KUKA KRL program: MyProgram_264().src

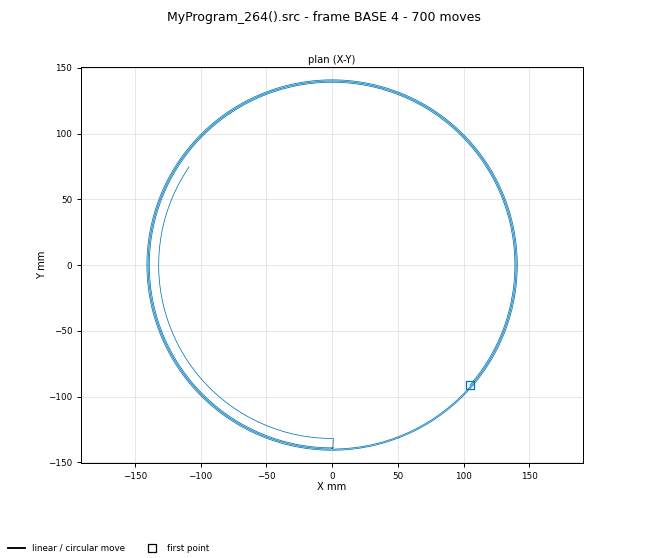
[picture p0: tool path of MyProgram_264().src in frame BASE 4, 700 of 700 moves have a stored position in this frame; points joined in program order, loops and branches not executed]
&ACCESS RVP
&REL 1
&PARAM TEMPLATE = C:\KRC\Roboter\Template\vorgabe
&PARAM EDITMASK = *
DEF MyProgram_264()
; ---- Setting reference (Base) ----
$BASE = BASE_DATA[4]

; --------------------------
; ---- Setting tool (TCP) ----
$TOOL = TOOL_DATA[3]
; --------------------------

$VEL.CP = VEL_APROX_PRINT
Startdeposition()
$VEL.CP = VEL_PRINT
LIN {X 104.7869,Y -91.2895,Z 168,A -38.7175,B 9.9687,C 0.2931,E1 10.0953,E2 489.8087} C_DIS
LIN {X 108.3715,Y -87.0044,Z 168,A -36.6212,B 9.9688,C 0.2929,E1 10.0989,E2 487.737} C_DIS
LIN {X 111.1205,Y -83.4649,Z 168,A -34.5628,B 9.9691,C 0.2832,E1 10.1024,E2 485.6491} C_DIS
LIN {X 113.1517,Y -80.6895,Z 168,A -32.7499,B 9.9694,C 0.2697,E1 10.1055,E2 483.7829} C_DIS
LIN {X 116.399,Y -75.9304,Z 168,A -31.0627,B 9.9691,C 0.2812,E1 10.1079,E2 482.1831} C_DIS
LIN {X 118.3407,Y -72.8666,Z 168,A -29.4296,B 9.9693,C 0.2739,E1 10.1104,E2 480.5305} C_DIS
LIN {X 120.9717,Y -68.4109,Z 168,A -27.417,B 9.9694,C 0.2715,E1 10.1131,E2 478.5313} C_DIS
LIN {X 123.1966,Y -64.3133,Z 168,A -24.8855,B 9.9699,C 0.2509,E1 10.1165,E2 475.918} C_DIS
LIN {X 125.8704,Y -58.9115,Z 168,A -23.1595,B 9.9696,C 0.2636,E1 10.1185,E2 474.2886} C_DIS
LIN {X 127.3983,Y -55.528,Z 168,A -21.7568,B 9.9696,C 0.2626,E1 10.1201,E2 472.9008} C_DIS
LIN {X 128.707,Y -52.4242,Z 168,A -20.3371,B 9.9698,C 0.2581,E1 10.1216,E2 471.4756} C_DIS
LIN {X 130.4635,Y -47.89,Z 168,A -18.2188,B 9.97,C 0.2496,E1 10.1237,E2 469.3404} C_DIS
LIN {X 131.6831,Y -44.4232,Z 168,A -16.8072,B 9.97,C 0.248,E1 10.125,E2 467.9405} C_DIS
LIN {X 132.7574,Y -41.1001,Z 168,A -15.3867,B 9.97,C 0.2445,E1 10.1262,E2 466.521} C_DIS
LIN {X 134.004,Y -36.8358,Z 168,A -13.5572,B 9.9702,C 0.2393,E1 10.1276,E2 464.6898} C_DIS
LIN {X 135.3311,Y -31.6154,Z 168,A -11.3086,B 9.9704,C 0.2323,E1 10.1291,E2 462.4352} C_DIS
LIN {X 136.0558,Y -28.3338,Z 168,A -9.341,B 9.9708,C 0.2134,E1 10.1302,E2 460.3905} C_DIS
LIN {X 137.1037,Y -22.7202,Z 168,A -8.0736,B 9.9703,C 0.2343,E1 10.1308,E2 459.2616} C_DIS
LIN {X 137.4864,Y -20.2859,Z 168,A -6.7394,B 9.9706,C 0.2233,E1 10.1313,E2 457.8854} C_DIS
LIN {X 137.9944,Y -16.4673,Z 168,A -5.1719,B 9.9706,C 0.2192,E1 10.1319,E2 456.3189} C_DIS
LIN {X 138.5607,Y -10.7209,Z 168,A -2.595,B 9.9709,C 0.2073,E1 10.1325,E2 453.7142} C_DIS
LIN {X 138.8592,Y -5.6425,Z 168,A -0.7367,B 9.9709,C 0.2073,E1 10.1328,E2 451.8846} C_DIS
LIN {X 138.9611,Y -1.9096,Z 168,A 0.6796,B 9.9709,C 0.2059,E1 10.1328,E2 450.4827} C_DIS
LIN {X 138.9263,Y 3.6331,Z 168,A 3.0218,B 9.9711,C 0.1978,E1 10.1328,E2 448.1311} C_DIS
LIN {X 138.6111,Y 10.0308,Z 168,A 5.6741,B 9.9713,C 0.1898,E1 10.1324,E2 445.4748} C_DIS
LIN {X 138.3396,Y 13.2584,Z 168,A 7.4808,B 9.9716,C 0.1739,E1 10.1319,E2 443.606} C_DIS
LIN {X 137.7917,Y 18.0849,Z 168,A 8.8238,B 9.9714,C 0.1849,E1 10.1314,E2 442.3462} C_DIS
LIN {X 137.0969,Y 22.761,Z 168,A 10.9205,B 9.9715,C 0.1756,E1 10.1305,E2 440.2289} C_DIS
LIN {X 136.0747,Y 28.2409,Z 168,A 13.3844,B 9.9717,C 0.1648,E1 10.1292,E2 437.7417} C_DIS
LIN {X 135.321,Y 31.66,Z 168,A 14.6274,B 9.9717,C 0.1658,E1 10.1284,E2 436.5233} C_DIS
LIN {X 134.3492,Y 35.5518,Z 168,A 16.1439,B 9.9717,C 0.1646,E1 10.1273,E2 435.023} C_DIS
LIN {X 133.4563,Y 38.7692,Z 168,A 17.4893,B 9.9717,C 0.1616,E1 10.1263,E2 433.6804} C_DIS
LIN {X 132.3926,Y 42.2583,Z 168,A 18.9598,B 9.9718,C 0.1582,E1 10.1251,E2 432.213} C_DIS
LIN {X 131.3467,Y 45.405,Z 168,A 20.2249,B 9.9718,C 0.157,E1 10.124,E2 430.9599} C_DIS
LIN {X 130.5672,Y 47.6024,Z 168,A 21.8935,B 9.9721,C 0.1366,E1 10.1223,E2 429.1998} C_DIS
LIN {X 128.6889,Y 52.4691,Z 168,A 23.0407,B 9.9719,C 0.156,E1 10.1212,E2 428.1795} C_DIS
LIN {X 127.1442,Y 56.1102,Z 168,A 25.0796,B 9.9721,C 0.1415,E1 10.1189,E2 426.0876} C_DIS
LIN {X 125.5425,Y 59.6045,Z 168,A 26.6572,B 9.9721,C 0.1375,E1 10.1171,E2 424.5098} C_DIS
LIN {X 123.808,Y 63.1275,Z 168,A 28.1243,B 9.9721,C 0.1371,E1 10.1152,E2 423.061} C_DIS
LIN {X 122.1696,Y 66.2478,Z 168,A 29.4062,B 9.9721,C 0.1377,E1 10.1136,E2 421.8} C_DIS
LIN {X 119.9358,Y 70.2099,Z 168,A 31.3397,B 9.9721,C 0.1316,E1 10.1109,E2 419.858} C_DIS
LIN {X 117.6886,Y 73.9159,Z 168,A 33.3363,B 9.9723,C 0.122,E1 10.1079,E2 417.8337} C_DIS
LIN {X 115.2813,Y 77.6165,Z 168,A 35.1156,B 9.9723,C 0.1186,E1 10.1052,E2 416.0585} C_DIS
LIN {X 112.6825,Y 81.3436,Z 168,A 36.9745,B 9.9724,C 0.1146,E1 10.1022,E2 414.2005} C_DIS
LIN {X 110.8525,Y 83.8201,Z 168,A 38.4939,B 9.9725,C 0.1055,E1 10.0996,E2 412.6485} C_DIS
LIN {X 108.4731,Y 86.8782,Z 168,A 39.6916,B 9.9725,C 0.1117,E1 10.0976,E2 411.5011} C_DIS
LIN {X 105.8164,Y 90.0942,Z 168,A 41.4849,B 9.9725,C 0.1061,E1 10.0944,E2 409.6976} C_DIS
LIN {X 99.6435,Y 96.8779,Z 168,A 45.2327,B 9.9725,C 0.099,E1 10.0873,E2 405.9528} C_DIS
LIN {X 97.1213,Y 99.4061,Z 168,A 46.8412,B 9.9726,C 0.0928,E1 10.084,E2 404.3264} C_DIS
LIN {X 93.1563,Y 103.1313,Z 168,A 48.9073,B 9.9726,C 0.0927,E1 10.0798,E2 402.2821} C_DIS
LIN {X 90.6095,Y 105.3754,Z 168,A 50.6855,B 9.9727,C 0.0809,E1 10.076,E2 400.4553} C_DIS
LIN {X 87.221,Y 108.1968,Z 168,A 52.1284,B 9.9727,C 0.0867,E1 10.0729,E2 399.0597} C_DIS
LIN {X 83.4306,Y 111.1464,Z 168,A 53.8675,B 9.9727,C 0.089,E1 10.0691,E2 397.3507} C_DIS
LIN {X 81.247,Y 112.7524,Z 168,A 55.195,B 9.9727,C 0.0821,E1 10.0661,E2 395.9964} C_DIS
LIN {X 77.5243,Y 115.344,Z 168,A 57.0601,B 9.9727,C 0.0792,E1 10.0618,E2 394.1316} C_DIS
LIN {X 73.7727,Y 117.7787,Z 168,A 58.8556,B 9.9727,C 0.0775,E1 10.0575,E2 392.3419} C_DIS
LIN {X 70.011,Y 120.053,Z 168,A 60.6788,B 9.9727,C 0.0746,E1 10.0532,E2 390.5172} C_DIS
LIN {X 66.8198,Y 121.8576,Z 168,A 62.1695,B 9.9727,C 0.073,E1 10.0495,E2 389.029} C_DIS
LIN {X 61.3179,Y 124.7143,Z 168,A 64.57,B 9.9727,C 0.0734,E1 10.0436,E2 386.6479} C_DIS
LIN {X 58.4874,Y 126.0665,Z 168,A 65.8378,B 9.9727,C 0.0724,E1 10.0404,E2 385.3833} C_DIS
LIN {X 55.3605,Y 127.4707,Z 168,A 67.2727,B 9.9728,C 0.0703,E1 10.0367,E2 383.9457} C_DIS
LIN {X 52.2262,Y 128.7868,Z 168,A 68.6604,B 9.9728,C 0.0691,E1 10.0332,E2 382.5599} C_DIS
LIN {X 48.8963,Y 130.0873,Z 168,A 70.0927,B 9.9728,C 0.0685,E1 10.0294,E2 381.1329} C_DIS
LIN {X 45.7955,Y 131.2113,Z 168,A 71.5098,B 9.9728,C 0.0659,E1 10.0257,E2 379.7088} C_DIS
LIN {X 42.4601,Y 132.3281,Z 168,A 72.9338,B 9.9728,C 0.0653,E1 10.0219,E2 378.2882} C_DIS
LIN {X 39.2358,Y 133.3197,Z 168,A 74.1058,B 9.9728,C 0.0691,E1 10.0189,E2 377.1439} C_DIS
LIN {X 35.492,Y 134.3651,Z 168,A 76.3709,B 9.9729,C 0.0529,E1 10.0125,E2 374.7958} C_DIS
LIN {X 31.4057,Y 135.3791,Z 168,A 77.701,B 9.9729,C 0.061,E1 10.0091,E2 373.5173} C_DIS
LIN {X 27.0023,Y 136.3268,Z 168,A 80.0388,B 9.9729,C 0.0492,E1 10.0025,E2 371.1194} C_DIS
LIN {X 22.5072,Y 137.1392,Z 168,A 81.6679,B 9.9729,C 0.0541,E1 9.9981,E2 369.5229} C_DIS
LIN {X 19.253,Y 137.634,Z 168,A 82.8687,B 9.9729,C 0.057,E1 9.9948,E2 368.3422} C_DIS
LIN {X 15.4145,Y 138.1171,Z 168,A 84.8657,B 9.9729,C 0.0477,E1 9.9892,E2 366.2951} C_DIS
LIN {X 10.7583,Y 138.558,Z 168,A 86.4757,B 9.9729,C 0.0543,E1 9.9848,E2 364.726} C_DIS
LIN {X 5.6517,Y 138.8588,Z 168,A 88.4161,B 9.9729,C 0.0578,E1 9.9794,E2 362.8077} C_DIS
LIN {X 1.3259,Y 138.9685,Z 168,A 90.5444,B 9.9729,C 0.0503,E1 9.9734,E2 360.6369} C_DIS
LIN {X -2.4839,Y 138.9515,Z 168,A 91.9187,B 9.9729,C 0.0547,E1 9.9696,E2 359.288} C_DIS
LIN {X -7.6751,Y 138.7632,Z 168,A 94.0131,B 9.9729,C 0.0561,E1 9.9638,E2 357.2007} C_DIS
LIN {X -11.7705,Y 138.4742,Z 168,A 96.3131,B 9.9729,C 0.0434,E1 9.9572,E2 354.8249} C_DIS
LIN {X -17.6085,Y 137.8542,Z 168,A 98.4749,B 9.9729,C 0.0499,E1 9.9513,E2 352.6973} C_DIS
LIN {X -22.0537,Y 137.2147,Z 168,A 99.978,B 9.9729,C 0.0583,E1 9.9473,E2 351.2392} C_DIS
LIN {X -26.5941,Y 136.406,Z 168,A 101.7752,B 9.9729,C 0.0616,E1 9.9424,E2 349.4562} C_DIS
LIN {X -30.5737,Y 135.5691,Z 168,A 103.454,B 9.9729,C 0.0626,E1 9.9378,E2 347.7783} C_DIS
LIN {X -34.2317,Y 134.6914,Z 168,A 104.9802,B 9.9729,C 0.0643,E1 9.9336,E2 346.2561} C_DIS
LIN {X -37.445,Y 133.8336,Z 168,A 106.4119,B 9.9729,C 0.0641,E1 9.9298,E2 344.8179} C_DIS
LIN {X -40.4898,Y 132.9442,Z 168,A 108.0789,B 9.9729,C 0.0578,E1 9.9252,E2 343.1067} C_DIS
LIN {X -44.2338,Y 131.7461,Z 168,A 109.3437,B 9.9729,C 0.0667,E1 9.922,E2 341.8879} C_DIS
LIN {X -48.1285,Y 130.3749,Z 168,A 110.9864,B 9.9729,C 0.0697,E1 9.9177,E2 340.2539} C_DIS
LIN {X -51.4358,Y 129.1054,Z 168,A 112.3928,B 9.9728,C 0.0724,E1 9.914,E2 338.8554} C_DIS
LIN {X -55.5497,Y 127.3889,Z 168,A 114.4516,B 9.9728,C 0.0701,E1 9.9087,E2 336.7705} C_DIS
LIN {X -59.5895,Y 125.5497,Z 168,A 116.094,B 9.9728,C 0.0762,E1 9.9046,E2 335.153} C_DIS
LIN {X -62.3414,Y 124.2079,Z 168,A 117.6958,B 9.9728,C 0.071,E1 9.9005,E2 333.5099} C_DIS
LIN {X -66.1173,Y 122.2404,Z 168,A 119.509,B 9.9728,C 0.0723,E1 9.896,E2 331.691} C_DIS
LIN {X -68.9786,Y 120.6484,Z 168,A 120.6619,B 9.9728,C 0.0783,E1 9.8933,E2 330.564} C_DIS
LIN {X -71.4953,Y 119.1748,Z 168,A 122.3694,B 9.9728,C 0.07,E1 9.8891,E2 328.7941} C_DIS
LIN {X -75.6051,Y 116.6102,Z 168,A 123.715,B 9.9727,C 0.0863,E1 9.8861,E2 327.5322} C_DIS
LIN {X -78.7988,Y 114.4764,Z 168,A 125.4857,B 9.9727,C 0.0852,E1 9.8819,E2 325.7395} C_DIS
LIN {X -82.4494,Y 111.8758,Z 168,A 127.1228,B 9.9727,C 0.0926,E1 9.8783,E2 324.1305} C_DIS
LIN {X -86.4838,Y 108.7871,Z 168,A 129.6992,B 9.9727,C 0.0869,E1 9.8725,E2 321.4958} C_DIS
LIN {X -89.1735,Y 106.5935,Z 168,A 130.916,B 9.9727,C 0.0938,E1 9.8699,E2 320.3074} C_DIS
LIN {X -92.5782,Y 103.6502,Z 168,A 132.755,B 9.9726,C 0.0978,E1 9.8661,E2 318.4723} C_DIS
LIN {X -96.5219,Y 99.9881,Z 168,A 135.3869,B 9.9726,C 0.0942,E1 9.8606,E2 315.7907} C_DIS
LIN {X -99.4725,Y 97.0537,Z 168,A 136.7519,B 9.9726,C 0.1047,E1 9.8581,E2 314.4716} C_DIS
LIN {X -102.5413,Y 93.8054,Z 168,A 138.3633,B 9.9724,C 0.1132,E1 9.8551,E2 312.891} C_DIS
LIN {X -105.8315,Y 90.0764,Z 168,A 141.0491,B 9.9725,C 0.1054,E1 9.85,E2 310.1276} C_DIS
LIN {X -108.4461,Y 86.9114,Z 168,A 142.4577,B 9.9725,C 0.1149,E1 9.8476,E2 308.7565} C_DIS
LIN {X -110.6702,Y 84.0616,Z 168,A 143.8995,B 9.9724,C 0.1193,E1 9.8452,E2 307.3224} C_DIS
LIN {X -113.7992,Y 79.7744,Z 168,A 146.1492,B 9.9724,C 0.1234,E1 9.8415,E2 305.0674} C_DIS
LIN {X -116.3521,Y 76.0026,Z 168,A 148.054,B 9.9723,C 0.1275,E1 9.8385,E2 303.1611} C_DIS
LIN {X -118.6956,Y 72.2884,Z 168,A 149.9103,B 9.9723,C 0.1311,E1 9.8358,E2 301.3011} C_DIS
LIN {X -120.9843,Y 68.3884,Z 168,A 151.8068,B 9.9722,C 0.1353,E1 9.8332,E2 299.4025} C_DIS
LIN {X -123.1081,Y 64.4819,Z 168,A 153.8724,B 9.9722,C 0.1356,E1 9.8304,E2 297.3095} C_DIS
LIN {X -124.7232,Y 61.2998,Z 168,A 155.1789,B 9.972,C 0.1426,E1 9.8288,E2 296.0254} C_DIS
LIN {X -127.0073,Y 56.4162,Z 168,A 157.3275,B 9.972,C 0.15,E1 9.8264,E2 293.8885} C_DIS
LIN {X -128.5481,Y 52.8162,Z 168,A 159.4017,B 9.972,C 0.1457,E1 9.8241,E2 291.7581} C_DIS
LIN {X -130.0853,Y 48.9017,Z 168,A 160.672,B 9.9718,C 0.1592,E1 9.8229,E2 290.5482} C_DIS
LIN {X -132.1241,Y 43.0961,Z 168,A 163.3195,B 9.9718,C 0.1642,E1 9.8205,E2 287.8896} C_DIS
LIN {X -133.3063,Y 39.2816,Z 168,A 164.9105,B 9.9716,C 0.1699,E1 9.8192,E2 286.3072} C_DIS
LIN {X -134.2142,Y 36.058,Z 168,A 166.3635,B 9.9716,C 0.1724,E1 9.8181,E2 284.8466} C_DIS
LIN {X -135.0793,Y 32.6675,Z 168,A 167.7655,B 9.9715,C 0.1773,E1 9.8172,E2 283.4512} C_DIS
LIN {X -135.8366,Y 29.3601,Z 168,A 169.1877,B 9.9715,C 0.1809,E1 9.8163,E2 282.0276} C_DIS
LIN {X -136.4454,Y 26.388,Z 168,A 170.5451,B 9.9715,C 0.1825,E1 9.8156,E2 280.6581} C_DIS
LIN {X -137.1353,Y 22.5308,Z 168,A 172.1893,B 9.9713,C 0.1866,E1 9.8148,E2 279.0119} C_DIS
LIN {X -137.7668,Y 18.2749,Z 168,A 173.9456,B 9.9713,C 0.1921,E1 9.8141,E2 277.2597} C_DIS
LIN {X -138.1801,Y 14.8292,Z 168,A 175.3528,B 9.9711,C 0.1967,E1 9.8137,E2 275.8569} C_DIS
LIN {X -138.6204,Y 9.9036,Z 168,A 177.2102,B 9.971,C 0.206,E1 9.8133,E2 274.0245} C_DIS
LIN {X -138.8726,Y 5.2979,Z 168,A 179.3932,B 9.971,C 0.2063,E1 9.813,E2 271.8079} C_DIS
LIN {X -138.9511,Y 2.5119,Z 168,A -178.8031,B 9.9711,C 0.1973,E1 9.8129,E2 269.9221} C_DIS
LIN {X -138.9457,Y -2.8364,Z 168,A -177.2929,B 9.9707,C 0.2169,E1 9.8129,E2 268.5026} C_DIS
LIN {X -138.7047,Y -8.6416,Z 168,A -174.7671,B 9.9707,C 0.2214,E1 9.8133,E2 265.9626} C_DIS
LIN {X -138.3646,Y -12.9984,Z 168,A -172.9482,B 9.9705,C 0.2263,E1 9.8137,E2 264.1432} C_DIS
LIN {X -137.9891,Y -16.5116,Z 168,A -171.4819,B 9.9705,C 0.2303,E1 9.8141,E2 262.677} C_DIS
LIN {X -137.4533,Y -20.5131,Z 168,A -169.6739,B 9.9704,C 0.2324,E1 9.8149,E2 260.8524} C_DIS
LIN {X -136.8786,Y -24.0426,Z 168,A -168.2662,B 9.9703,C 0.2379,E1 9.8155,E2 259.4545} C_DIS
LIN {X -136.2873,Y -27.1964,Z 168,A -166.9044,B 9.9702,C 0.2409,E1 9.8163,E2 258.0889} C_DIS
LIN {X -135.5229,Y -30.7758,Z 168,A -165.4066,B 9.9701,C 0.2454,E1 9.8172,E2 256.5938} C_DIS
LIN {X -134.672,Y -34.308,Z 168,A -163.9032,B 9.97,C 0.2495,E1 9.8182,E2 255.0909} C_DIS
LIN {X -133.92,Y -37.1362,Z 168,A -162.3001,B 9.97,C 0.2453,E1 9.8194,E2 253.4382} C_DIS
LIN {X -132.8591,Y -40.768,Z 168,A -161.1109,B 9.9698,C 0.2567,E1 9.8203,E2 252.2976} C_DIS
LIN {X -131.6541,Y -44.5101,Z 168,A -159.3701,B 9.9698,C 0.2588,E1 9.8219,E2 250.5428} C_DIS
LIN {X -130.2278,Y -48.5213,Z 168,A -157.5157,B 9.9697,C 0.2617,E1 9.8236,E2 248.6771} C_DIS
LIN {X -128.3545,Y -53.2798,Z 168,A -155.5113,B 9.9695,C 0.2693,E1 9.8257,E2 246.6875} C_DIS
LIN {X -126.9695,Y -56.5007,Z 168,A -154.0901,B 9.9693,C 0.2736,E1 9.8273,E2 245.2705} C_DIS
LIN {X -125.5352,Y -59.6198,Z 168,A -152.6233,B 9.9693,C 0.2763,E1 9.8291,E2 243.798} C_DIS
LIN {X -124.0044,Y -62.7419,Z 168,A -151.1771,B 9.9692,C 0.2797,E1 9.8309,E2 242.3512} C_DIS
LIN {X -122.2078,Y -66.1778,Z 168,A -149.4378,B 9.9692,C 0.281,E1 9.8332,E2 240.595} C_DIS
LIN {X -119.9592,Y -70.1707,Z 168,A -147.5406,B 9.969,C 0.2855,E1 9.8358,E2 238.698} C_DIS
LIN {X -117.5827,Y -74.0837,Z 168,A -145.6598,B 9.9689,C 0.2902,E1 9.8386,E2 236.8191} C_DIS
LIN {X -115.2184,Y -77.71,Z 168,A -143.8229,B 9.9688,C 0.2935,E1 9.8414,E2 234.9765} C_DIS
LIN {X -112.5662,Y -81.5042,Z 168,A -142.027,B 9.9686,C 0.3001,E1 9.8443,E2 233.1961} C_DIS
LIN {X -110.0316,Y -84.8953,Z 168,A -140.3109,B 9.9685,C 0.3046,E1 9.8472,E2 231.4847} C_DIS
LIN {X -107.8706,Y -87.6252,Z 168,A -138.6725,B 9.9685,C 0.3038,E1 9.8501,E2 229.8208} C_DIS
LIN {X -103.7204,Y -92.4993,Z 168,A -135.7389,B 9.9685,C 0.3035,E1 9.8555,E2 226.8505} C_DIS
LIN {X -101.1547,Y -95.2985,Z 168,A -134.4399,B 9.9682,C 0.3121,E1 9.858,E2 225.5864} C_DIS
LIN {X -97.8845,Y -98.6544,Z 168,A -132.4981,B 9.9682,C 0.3157,E1 9.8618,E2 223.644} C_DIS
LIN {X -94.6627,Y -101.7499,Z 168,A -130.6386,B 9.968,C 0.3189,E1 9.8655,E2 221.783} C_DIS
LIN {X -91.8147,Y -104.3272,Z 168,A -128.9762,B 9.968,C 0.3202,E1 9.869,E2 220.1109} C_DIS
LIN {X -88.6264,Y -107.0487,Z 168,A -127.3089,B 9.9678,C 0.3246,E1 9.8726,E2 218.4519} C_DIS
LIN {X -85.2071,Y -109.7899,Z 168,A -125.4605,B 9.9678,C 0.3268,E1 9.8767,E2 216.5985} C_DIS
LIN {X -81.5915,Y -112.5029,Z 168,A -123.5971,B 9.9677,C 0.3299,E1 9.8808,E2 214.7355} C_DIS
LIN {X -77.8514,Y -115.1227,Z 168,A -121.7099,B 9.9676,C 0.3327,E1 9.8852,E2 212.8481} C_DIS
LIN {X -74.0236,Y -117.6206,Z 168,A -119.7892,B 9.9675,C 0.3347,E1 9.8897,E2 210.9229} C_DIS
LIN {X -70.0766,Y -120.0145,Z 168,A -117.8536,B 9.9675,C 0.3367,E1 9.8944,E2 208.9834} C_DIS
LIN {X -66.2604,Y -122.1627,Z 168,A -116.0362,B 9.9674,C 0.3388,E1 9.8988,E2 207.1645} C_DIS
LIN {X -63.1572,Y -123.7929,Z 168,A -114.6931,B 9.9672,C 0.3427,E1 9.9021,E2 205.8346} C_DIS
LIN {X -60.076,Y -125.3173,Z 168,A -113.2527,B 9.9672,C 0.3439,E1 9.9057,E2 204.3912} C_DIS
LIN {X -56.99,Y -126.7507,Z 168,A -111.8516,B 9.9672,C 0.3455,E1 9.9093,E2 202.9904} C_DIS
LIN {X -53.7974,Y -128.1383,Z 168,A -110.4369,B 9.9671,C 0.3474,E1 9.9129,E2 201.5782} C_DIS
LIN {X -50.5951,Y -129.4369,Z 168,A -108.9413,B 9.9671,C 0.3473,E1 9.9168,E2 200.0733} C_DIS
LIN {X -47.4345,Y -130.6277,Z 168,A -107.6075,B 9.967,C 0.3498,E1 9.9203,E2 198.7469} C_DIS
LIN {X -44.5463,Y -131.642,Z 168,A -106.2701,B 9.967,C 0.3492,E1 9.9239,E2 197.3997} C_DIS
LIN {X -41.1194,Y -132.7515,Z 168,A -104.4795,B 9.9672,C 0.3437,E1 9.9287,E2 195.5691} C_DIS
LIN {X -37.6879,Y -133.7657,Z 168,A -102.9081,B 9.9672,C 0.3426,E1 9.933,E2 193.9848} C_DIS
LIN {X -33.6552,Y -134.8377,Z 168,A -101.5008,B 9.967,C 0.3505,E1 9.9367,E2 192.6181} C_DIS
LIN {X -30.6389,Y -135.5542,Z 168,A -99.7171,B 9.9673,C 0.34,E1 9.9418,E2 190.7679} C_DIS
LIN {X -25.5906,Y -136.5979,Z 168,A -98.0857,B 9.9669,C 0.3518,E1 9.946,E2 189.2006} C_DIS
LIN {X -21.523,Y -137.2969,Z 168,A -96.505,B 9.9668,C 0.3551,E1 9.9504,E2 187.6351} C_DIS
LIN {X -18.216,Y -137.7745,Z 168,A -94.7786,B 9.9671,C 0.3477,E1 9.9553,E2 185.8627} C_DIS
LIN {X -14.6133,Y -138.2033,Z 168,A -93.4629,B 9.9669,C 0.352,E1 9.9589,E2 184.57} C_DIS
LIN {X -10.1404,Y -138.6031,Z 168,A -91.8449,B 9.9667,C 0.3574,E1 9.9633,E2 182.9817} C_DIS
LIN {X -7.0454,Y -138.7949,Z 168,A -90.4579,B 9.9668,C 0.355,E1 9.9672,E2 181.58} C_DIS
LIN {X -3.3684,Y -138.9337,Z 168,A -88.765,B 9.9669,C 0.351,E1 9.972,E2 179.8635} C_DIS
LIN {X 0.9911,Y -138.96,Z 168,A -87.4345,B 9.9666,C 0.3613,E1 9.9755,E2 178.5925} C_DIS
Enddeposition()
LIN {X 0.9911,Y -138.96,Z 168,A -87.4345,B 9.9666,C 0.3613,E1 9.9755,E2 178.5925} C_DIS
Startdeposition()
$VEL.CP = VEL_PRINT
LIN {X -1.4023,Y -139.882,Z 168,A -88.8873,B 9.9659,C 0.378,E1 9.9712,E2 180.1419} C_DIS
LIN {X -5.538,Y -139.778,Z 168,A -90.4696,B 9.966,C 0.3756,E1 9.9668,E2 181.7105} C_DIS
LIN {X -8.7861,Y -139.6115,Z 168,A -91.8405,B 9.966,C 0.3764,E1 9.963,E2 183.087} C_DIS
LIN {X -13.6462,Y -139.2206,Z 168,A -93.8637,B 9.966,C 0.3767,E1 9.9573,E2 185.1143} C_DIS
LIN {X -17.7268,Y -138.7605,Z 168,A -95.3215,B 9.9662,C 0.3714,E1 9.9534,E2 186.5437} C_DIS
LIN {X -20.0407,Y -138.4447,Z 168,A -96.4484,B 9.9661,C 0.3749,E1 9.9502,E2 187.693} C_DIS
LIN {X -23.5763,Y -137.8875,Z 168,A -97.8514,B 9.9661,C 0.373,E1 9.9463,E2 189.0883} C_DIS
LIN {X -26.9584,Y -137.2669,Z 168,A -99.2952,B 9.9661,C 0.3732,E1 9.9424,E2 190.5371} C_DIS
LIN {X -30.6958,Y -136.4786,Z 168,A -100.726,B 9.9663,C 0.3695,E1 9.9385,E2 191.951} C_DIS
LIN {X -33.2645,Y -135.8756,Z 168,A -103.2247,B 9.9651,C 0.3993,E1 9.9313,E2 194.6315} C_DIS
LIN {X -41.6421,Y -133.5474,Z 168,A -105.5327,B 9.9662,C 0.3701,E1 9.9255,E2 196.7802} C_DIS
LIN {X -45.6049,Y -132.2447,Z 168,A -107.2791,B 9.9662,C 0.3695,E1 9.9208,E2 198.5317} C_DIS
LIN {X -49.3445,Y -130.8954,Z 168,A -108.9184,B 9.9662,C 0.3683,E1 9.9165,E2 200.1725} C_DIS
LIN {X -52.5844,Y -129.6278,Z 168,A -110.3296,B 9.9664,C 0.3666,E1 9.9129,E2 201.5821} C_DIS
LIN {X -55.7525,Y -128.297,Z 168,A -111.7289,B 9.9664,C 0.365,E1 9.9093,E2 202.9804} C_DIS
LIN {X -59.0082,Y -126.8327,Z 168,A -113.2206,B 9.9664,C 0.364,E1 9.9055,E2 204.4759} C_DIS
LIN {X -62.2547,Y -125.2713,Z 168,A -114.7585,B 9.9664,C 0.3636,E1 9.9016,E2 206.0219} C_DIS
LIN {X -66.4519,Y -123.0982,Z 168,A -116.7177,B 9.9665,C 0.3617,E1 9.8968,E2 207.984} C_DIS
LIN {X -70.2359,Y -120.9789,Z 168,A -118.4998,B 9.9666,C 0.3594,E1 9.8924,E2 209.7667} C_DIS
LIN {X -73.953,Y -118.743,Z 168,A -120.2924,B 9.9666,C 0.3572,E1 9.8882,E2 211.5611} C_DIS
LIN {X -77.5468,Y -116.4279,Z 168,A -122.0861,B 9.9668,C 0.3555,E1 9.884,E2 213.3602} C_DIS
LIN {X -81.3861,Y -113.7772,Z 168,A -123.9753,B 9.9668,C 0.352,E1 9.8797,E2 215.2462} C_DIS
LIN {X -84.7126,Y -111.3231,Z 168,A -125.7393,B 9.9669,C 0.3506,E1 9.8757,E2 217.0189} C_DIS
LIN {X -88.2981,Y -108.501,Z 168,A -127.6222,B 9.967,C 0.3477,E1 9.8716,E2 218.9032} C_DIS
LIN {X -93.4849,Y -104.0652,Z 168,A -130.393,B 9.9672,C 0.3421,E1 9.8658,E2 221.67} C_DIS
LIN {X -96.7853,Y -101.0029,Z 168,A -132.2824,B 9.9673,C 0.3394,E1 9.8619,E2 223.5646} C_DIS
LIN {X -100.4272,Y -97.3823,Z 168,A -134.2291,B 9.9676,C 0.3321,E1 9.8581,E2 225.4905} C_DIS
LIN {X -107.0765,Y -90.0199,Z 168,A -138.1499,B 9.9679,C 0.3208,E1 9.8509,E2 229.3915} C_DIS
LIN {X -110.4439,Y -85.8552,Z 168,A -141.092,B 9.9676,C 0.3307,E1 9.8456,E2 232.4282} C_DIS
LIN {X -112.9995,Y -82.4636,Z 168,A -142.3318,B 9.968,C 0.317,E1 9.8436,E2 233.6036} C_DIS
LIN {X -115.0902,Y -79.5197,Z 168,A -143.9424,B 9.968,C 0.3161,E1 9.841,E2 235.2302} C_DIS
LIN {X -117.5104,Y -75.897,Z 168,A -145.7789,B 9.9682,C 0.3129,E1 9.8382,E2 237.0723} C_DIS
LIN {X -119.9217,Y -72.0271,Z 168,A -147.7017,B 9.9682,C 0.3094,E1 9.8354,E2 239.001} C_DIS
LIN {X -122.2189,Y -68.0559,Z 168,A -149.5371,B 9.9684,C 0.3039,E1 9.8328,E2 240.8297} C_DIS
LIN {X -124.0221,Y -64.7073,Z 168,A -151.091,B 9.9686,C 0.2999,E1 9.8308,E2 242.382} C_DIS
LIN {X -125.5767,Y -61.6357,Z 168,A -152.509,B 9.9686,C 0.2964,E1 9.829,E2 243.8001} C_DIS
LIN {X -127.1223,Y -58.3818,Z 168,A -154.0006,B 9.9688,C 0.2929,E1 9.8273,E2 245.2927} C_DIS
LIN {X -128.531,Y -55.2114,Z 168,A -155.4632,B 9.9688,C 0.2899,E1 9.8256,E2 246.7595} C_DIS
LIN {X -130.157,Y -51.2636,Z 168,A -157.1198,B 9.969,C 0.2835,E1 9.8239,E2 248.4032} C_DIS
LIN {X -131.1125,Y -48.7649,Z 168,A -158.3166,B 9.969,C 0.2825,E1 9.8227,E2 249.612} C_DIS
LIN {X -132.3803,Y -45.2137,Z 168,A -159.8632,B 9.9692,C 0.2783,E1 9.8213,E2 251.1577} C_DIS
LIN {X -133.4731,Y -41.8794,Z 168,A -161.324,B 9.9692,C 0.2748,E1 9.82,E2 252.6203} C_DIS
LIN {X -134.2219,Y -39.4072,Z 168,A -162.4853,B 9.9693,C 0.2738,E1 9.8191,E2 253.7938} C_DIS
LIN {X -135.2052,Y -35.889,Z 168,A -163.9543,B 9.9694,C 0.2691,E1 9.818,E2 255.2582} C_DIS
LIN {X -136.156,Y -32.1012,Z 168,A -165.6438,B 9.9695,C 0.2664,E1 9.8169,E2 256.9578} C_DIS
LIN {X -137.0477,Y -28.0433,Z 168,A -167.3693,B 9.9696,C 0.262,E1 9.8159,E2 258.6848} C_DIS
LIN {X -137.884,Y -23.5971,Z 168,A -169.2693,B 9.9697,C 0.2576,E1 9.815,E2 260.5891} C_DIS
LIN {X -138.5706,Y -19.1596,Z 168,A -171.0115,B 9.9699,C 0.2505,E1 9.8142,E2 262.3174} C_DIS
LIN {X -138.9472,Y -16.1966,Z 168,A -172.3599,B 9.9699,C 0.2493,E1 9.8138,E2 263.6804} C_DIS
LIN {X -139.4144,Y -11.4981,Z 168,A -174.2048,B 9.9701,C 0.242,E1 9.8133,E2 265.5123} C_DIS
LIN {X -139.8329,Y -3.9121,Z 168,A -178.3598,B 9.9699,C 0.2523,E1 9.8128,E2 269.7949} C_DIS
LIN {X -139.8553,Y 3.1032,Z 168,A 178.8698,B 9.9701,C 0.242,E1 9.813,E2 272.5497} C_DIS
LIN {X -139.5865,Y 9.1909,Z 168,A 177.2072,B 9.9706,C 0.2193,E1 9.8132,E2 274.1056} C_DIS
LIN {X -139.0623,Y 15.1737,Z 168,A 174.6787,B 9.9708,C 0.2134,E1 9.8139,E2 276.6402} C_DIS
LIN {X -138.6396,Y 18.649,Z 168,A 173.2033,B 9.9708,C 0.2101,E1 9.8144,E2 278.1194} C_DIS
LIN {X -138.0188,Y 22.7896,Z 168,A 171.3223,B 9.9708,C 0.2082,E1 9.8152,E2 280.0195} C_DIS
LIN {X -137.3108,Y 26.7289,Z 168,A 169.7506,B 9.971,C 0.2022,E1 9.816,E2 281.581} C_DIS
LIN {X -136.6672,Y 29.8436,Z 168,A 168.4553,B 9.971,C 0.1983,E1 9.8168,E2 282.874} C_DIS
LIN {X -135.9793,Y 32.8343,Z 168,A 167.1881,B 9.9711,C 0.1949,E1 9.8176,E2 284.1411} C_DIS
LIN {X -135.12,Y 36.2084,Z 168,A 165.7403,B 9.9712,C 0.1913,E1 9.8186,E2 285.5902} C_DIS
LIN {X -134.268,Y 39.2497,Z 168,A 164.3992,B 9.9712,C 0.1885,E1 9.8197,E2 286.9358} C_DIS
LIN {X -133.1958,Y 42.7475,Z 168,A 162.9069,B 9.9713,C 0.1842,E1 9.8209,E2 288.4258} C_DIS
LIN {X -132.0627,Y 46.13,Z 168,A 161.4219,B 9.9714,C 0.1806,E1 9.8223,E2 289.9122} C_DIS
LIN {X -130.6792,Y 49.9201,Z 168,A 159.6293,B 9.9714,C 0.1787,E1 9.824,E2 291.7205} C_DIS
LIN {X -129.2527,Y 53.5009,Z 168,A 158.3113,B 9.9716,C 0.1695,E1 9.8254,E2 293.0041} C_DIS
LIN {X -127.8775,Y 56.7093,Z 168,A 156.5179,B 9.9716,C 0.1725,E1 9.8274,E2 294.8415} C_DIS
LIN {X -125.7458,Y 61.291,Z 168,A 154.2174,B 9.9716,C 0.1713,E1 9.8302,E2 297.1685} C_DIS
LIN {X -124.0271,Y 64.6977,Z 168,A 153.0806,B 9.9718,C 0.1592,E1 9.8316,E2 298.2505} C_DIS
LIN {X -122.1434,Y 68.1916,Z 168,A 151.2429,B 9.9718,C 0.159,E1 9.8341,E2 300.113} C_DIS
LIN {X -119.8262,Y 72.185,Z 168,A 149.3409,B 9.9718,C 0.1544,E1 9.8368,E2 302.0143} C_DIS
LIN {X -117.3414,Y 76.1573,Z 168,A 147.4193,B 9.9719,C 0.1497,E1 9.8397,E2 303.9342} C_DIS
LIN {X -114.7062,Y 80.0717,Z 168,A 145.1196,B 9.9719,C 0.1519,E1 9.8434,E2 306.2774} C_DIS
LIN {X -112.3104,Y 83.3988,Z 168,A 144.0752,B 9.9721,C 0.1358,E1 9.845,E2 307.241} C_DIS
LIN {X -110.4865,Y 85.8003,Z 168,A 142.5209,B 9.9721,C 0.139,E1 9.8477,E2 308.8339} C_DIS
LIN {X -105.8547,Y 91.4536,Z 168,A 139.5006,B 9.9721,C 0.1328,E1 9.8531,E2 311.8545} C_DIS
LIN {X -103.1883,Y 94.4521,Z 168,A 137.816,B 9.9721,C 0.1299,E1 9.8563,E2 313.5424} C_DIS
LIN {X -100.0915,Y 97.7278,Z 168,A 135.9748,B 9.9722,C 0.1259,E1 9.8598,E2 315.3812} C_DIS
LIN {X -96.8068,Y 100.9823,Z 168,A 134.058,B 9.9722,C 0.1224,E1 9.8636,E2 317.2989} C_DIS
LIN {X -93.6776,Y 103.8924,Z 168,A 132.2329,B 9.9723,C 0.1204,E1 9.8674,E2 319.1316} C_DIS
LIN {X -90.2691,Y 106.8673,Z 168,A 130.3948,B 9.9723,C 0.1165,E1 9.8713,E2 320.9659} C_DIS
LIN {X -86.6616,Y 109.8126,Z 168,A 128.5093,B 9.9724,C 0.1125,E1 9.8754,E2 322.8469} C_DIS
LIN {X -84.3079,Y 111.6294,Z 168,A 127.2407,B 9.9724,C 0.1113,E1 9.8782,E2 324.1207} C_DIS
LIN {X -80.5091,Y 114.3995,Z 168,A 125.312,B 9.9724,C 0.108,E1 9.8826,E2 326.0479} C_DIS
LIN {X -76.7483,Y 116.9559,Z 168,A 123.4257,B 9.9724,C 0.1054,E1 9.887,E2 327.9354} C_DIS
LIN {X -71.7804,Y 120.0689,Z 168,A 121.2379,B 9.9726,C 0.0974,E1 9.8921,E2 330.0946} C_DIS
LIN {X -66.2749,Y 123.1933,Z 168,A 118.4982,B 9.9726,C 0.0966,E1 9.8988,E2 332.8504} C_DIS
LIN {X -61.0677,Y 125.8565,Z 168,A 116.0778,B 9.9726,C 0.0938,E1 9.9049,E2 335.2719} C_DIS
LIN {X -58.4483,Y 127.0916,Z 168,A 114.8595,B 9.9726,C 0.093,E1 9.9079,E2 336.4931} C_DIS
LIN {X -54.9506,Y 128.6437,Z 168,A 113.2188,B 9.9726,C 0.0926,E1 9.9122,E2 338.1417} C_DIS
LIN {X -51.3521,Y 130.1226,Z 168,A 111.7524,B 9.9726,C 0.0882,E1 9.9159,E2 339.5911} C_DIS
LIN {X -48.6083,Y 131.1712,Z 168,A 110.4429,B 9.9726,C 0.0891,E1 9.9194,E2 340.9129} C_DIS
LIN {X -45.3502,Y 132.333,Z 168,A 109.0887,B 9.9726,C 0.0864,E1 9.9229,E2 342.2582} C_DIS
LIN {X -41.9211,Y 133.4598,Z 168,A 107.5719,B 9.9726,C 0.0858,E1 9.927,E2 343.7788} C_DIS
LIN {X -38.6311,Y 134.4491,Z 168,A 106.193,B 9.9726,C 0.084,E1 9.9306,E2 345.1532} C_DIS
LIN {X -35.6928,Y 135.2575,Z 168,A 104.8938,B 9.9726,C 0.084,E1 9.9342,E2 346.4578} C_DIS
LIN {X -31.7363,Y 136.2411,Z 168,A 103.18,B 9.9726,C 0.0838,E1 9.9388,E2 348.1759} C_DIS
LIN {X -25.6318,Y 137.5206,Z 168,A 100.7393,B 9.9727,C 0.0799,E1 9.9455,E2 350.6008} C_DIS
LIN {X -18.4068,Y 138.6713,Z 168,A 97.4241,B 9.9727,C 0.0852,E1 9.9547,E2 353.9538} C_DIS
LIN {X -11.8435,Y 139.3853,Z 168,A 94.8917,B 9.9727,C 0.0806,E1 9.9617,E2 356.4634} C_DIS
LIN {X -7.2739,Y 139.6986,Z 168,A 93.0204,B 9.9727,C 0.0801,E1 9.9669,E2 358.3331} C_DIS
LIN {X -3.5355,Y 139.8434,Z 168,A 91.3893,B 9.9727,C 0.0821,E1 9.9715,E2 359.9757} C_DIS
LIN {X 0.8977,Y 139.8848,Z 168,A 89.6991,B 9.9727,C 0.0793,E1 9.9762,E2 361.6495} C_DIS
LIN {X 4.292,Y 139.8223,Z 168,A 88.273,B 9.9727,C 0.0801,E1 9.9802,E2 363.0794} C_DIS
LIN {X 8.1747,Y 139.6491,Z 168,A 86.6707,B 9.9727,C 0.0805,E1 9.9846,E2 364.6824} C_DIS
LIN {X 12.2876,Y 139.3478,Z 168,A 84.9422,B 9.9727,C 0.0817,E1 9.9895,E2 366.4151} C_DIS
LIN {X 16.6188,Y 138.8968,Z 168,A 83.2427,B 9.9727,C 0.0804,E1 9.9941,E2 368.1036} C_DIS
LIN {X 20.4841,Y 138.3813,Z 168,A 81.7085,B 9.9727,C 0.0796,E1 9.9984,E2 369.6295} C_DIS
LIN {X 23.1765,Y 137.9542,Z 168,A 80.4563,B 9.9727,C 0.0831,E1 10.0019,E2 370.8982} C_DIS
LIN {X 28.2408,Y 137.0075,Z 168,A 78.6269,B 9.9727,C 0.0779,E1 10.0068,E2 372.6919} C_DIS
LIN {X 31.4394,Y 136.3089,Z 168,A 76.0352,B 9.9725,C 0.1066,E1 10.0143,E2 375.4383} C_DIS
LIN {X 38.9644,Y 134.3515,Z 168,A 74.143,B 9.9727,C 0.0801,E1 10.0189,E2 377.1698} C_DIS
LIN {X 43.0594,Y 133.0961,Z 168,A 72.2222,B 9.9727,C 0.0853,E1 10.0241,E2 379.1113} C_DIS
LIN {X 46.1462,Y 132.057,Z 168,A 70.8511,B 9.9727,C 0.0874,E1 10.0277,E2 380.4868} C_DIS
LIN {X 49.3692,Y 130.8862,Z 168,A 69.522,B 9.9727,C 0.087,E1 10.0312,E2 381.8064} C_DIS
LIN {X 52.4445,Y 129.6842,Z 168,A 68.1976,B 9.9727,C 0.0878,E1 10.0346,E2 383.1272} C_DIS
LIN {X 55.7419,Y 128.3016,Z 168,A 66.6513,B 9.9727,C 0.0913,E1 10.0386,E2 384.6836} C_DIS
LIN {X 59.8388,Y 126.4435,Z 168,A 64.6944,B 9.9726,C 0.0961,E1 10.0436,E2 386.6549} C_DIS
LIN {X 67.4733,Y 122.5415,Z 168,A 61.357,B 9.9726,C 0.0967,E1 10.0518,E2 389.9707} C_DIS
LIN {X 71.1425,Y 120.4484,Z 168,A 59.5977,B 9.9726,C 0.0998,E1 10.0561,E2 391.7339} C_DIS
LIN {X 74.7791,Y 118.2246,Z 168,A 57.8591,B 9.9726,C 0.1023,E1 10.0602,E2 393.4717} C_DIS
LIN {X 78.4689,Y 115.8083,Z 168,A 55.941,B 9.9725,C 0.1078,E1 10.0647,E2 395.4041} C_DIS
LIN {X 81.9323,Y 113.3846,Z 168,A 54.2785,B 9.9725,C 0.109,E1 10.0684,E2 397.0583} C_DIS
LIN {X 85.7147,Y 110.5529,Z 168,A 52.4037,B 9.9725,C 0.1109,E1 10.0726,E2 398.926} C_DIS
LIN {X 89.3607,Y 107.6273,Z 168,A 50.403,B 9.9724,C 0.1165,E1 10.0769,E2 400.938} C_DIS
LIN {X 93.1017,Y 104.4083,Z 168,A 48.4643,B 9.9724,C 0.1183,E1 10.081,E2 402.8669} C_DIS
LIN {X 96.5709,Y 101.2078,Z 168,A 46.651,B 9.9724,C 0.1192,E1 10.0847,E2 404.6656} C_DIS
LIN {X 99.5565,Y 98.2733,Z 168,A 44.9078,B 9.9723,C 0.1234,E1 10.0881,E2 406.4131} C_DIS
LIN {X 102.5803,Y 95.1121,Z 168,A 42.9324,B 9.9722,C 0.1316,E1 10.0919,E2 408.4123} C_DIS
LIN {X 104.7393,Y 92.7288,Z 168,A 41.8949,B 9.9722,C 0.1276,E1 10.0938,E2 409.4151} C_DIS
LIN {X 107.3905,Y 89.6457,Z 168,A 40.2073,B 9.9722,C 0.1318,E1 10.0969,E2 411.1063} C_DIS
LIN {X 110.1153,Y 86.2762,Z 168,A 38.2997,B 9.9721,C 0.139,E1 10.1002,E2 413.0315} C_DIS
LIN {X 113.0732,Y 82.3621,Z 168,A 36.4053,B 9.9721,C 0.1409,E1 10.1033,E2 414.9124} C_DIS
LIN {X 115.6364,Y 78.7229,Z 168,A 34.4344,B 9.9719,C 0.1488,E1 10.1065,E2 416.903} C_DIS
LIN {X 117.4314,Y 76.0188,Z 168,A 32.4121,B 9.9716,C 0.1689,E1 10.1097,E2 419.0127} C_DIS
LIN {X 121.2031,Y 69.8487,Z 168,A 30.2979,B 9.9718,C 0.1556,E1 10.1125,E2 421.0225} C_DIS
LIN {X 123.0274,Y 66.5837,Z 168,A 28.8477,B 9.9718,C 0.1575,E1 10.1144,E2 422.4635} C_DIS
LIN {X 124.7877,Y 63.2178,Z 168,A 27.3858,B 9.9718,C 0.1591,E1 10.1163,E2 423.9143} C_DIS
LIN {X 127.0677,Y 58.5,Z 168,A 25.29,B 9.9718,C 0.1635,E1 10.1188,E2 426.0053} C_DIS
LIN {X 128.5761,Y 55.107,Z 168,A 23.2651,B 9.9714,C 0.18,E1 10.1211,E2 428.095} C_DIS
LIN {X 130.3606,Y 50.7398,Z 168,A 21.7924,B 9.9715,C 0.1738,E1 10.1226,E2 429.511} C_DIS
LIN {X 131.7747,Y 46.948,Z 168,A 20.2933,B 9.9715,C 0.1744,E1 10.124,E2 430.9913} C_DIS
LIN {X 132.87,Y 43.7517,Z 168,A 18.8866,B 9.9715,C 0.1788,E1 10.1252,E2 432.402} C_DIS
LIN {X 133.9216,Y 40.4194,Z 168,A 17.5117,B 9.9715,C 0.1813,E1 10.1264,E2 433.7708} C_DIS
LIN {X 134.7557,Y 37.5413,Z 168,A 16.2804,B 9.9713,C 0.1848,E1 10.1273,E2 435.0036} C_DIS
LIN {X 135.5394,Y 34.6057,Z 168,A 15.0395,B 9.9713,C 0.1883,E1 10.1282,E2 436.2451} C_DIS
LIN {X 136.9335,Y 28.6043,Z 168,A 12.6159,B 9.9712,C 0.1929,E1 10.1297,E2 438.6583} C_DIS
LIN {X 137.7189,Y 24.5353,Z 168,A 10.8518,B 9.9711,C 0.1994,E1 10.1306,E2 440.4323} C_DIS
LIN {X 138.4094,Y 20.2872,Z 168,A 8.7746,B 9.9708,C 0.2124,E1 10.1315,E2 442.5511} C_DIS
LIN {X 138.9082,Y 16.523,Z 168,A 7.5445,B 9.9708,C 0.2087,E1 10.1319,E2 443.7412} C_DIS
LIN {X 139.3327,Y 12.466,Z 168,A 6.0373,B 9.9708,C 0.2095,E1 10.1323,E2 445.2292} C_DIS
LIN {X 139.5796,Y 9.3033,Z 168,A 4.483,B 9.9706,C 0.2197,E1 10.1326,E2 446.8172} C_DIS
LIN {X 139.7936,Y 5.1381,Z 168,A 2.9548,B 9.9706,C 0.2201,E1 10.1328,E2 448.3241} C_DIS
LIN {X 139.8868,Y 0.7373,Z 168,A 1.2013,B 9.9706,C 0.2241,E1 10.1328,E2 450.073} C_DIS
LIN {X 139.8543,Y -3.1419,Z 168,A -0.3545,B 9.9705,C 0.2279,E1 10.1328,E2 451.6262} C_DIS
LIN {X 139.705,Y -7.1457,Z 168,A -2.0144,B 9.9703,C 0.2332,E1 10.1326,E2 453.29} C_DIS
LIN {X 139.4001,Y -11.6674,Z 168,A -3.8142,B 9.9703,C 0.2372,E1 10.1322,E2 455.0845} C_DIS
LIN {X 139.0544,Y -15.2466,Z 168,A -5.1746,B 9.9703,C 0.2386,E1 10.1318,E2 456.432} C_DIS
LIN {X 138.5807,Y -19.0889,Z 168,A -6.8822,B 9.97,C 0.2464,E1 10.1312,E2 458.157} C_DIS
LIN {X 137.9596,Y -23.1443,Z 168,A -8.4829,B 9.97,C 0.2492,E1 10.1305,E2 459.7492} C_DIS
LIN {X 137.3071,Y -26.7482,Z 168,A -10.0172,B 9.9698,C 0.2544,E1 10.1297,E2 461.2895} C_DIS
LIN {X 136.3057,Y -31.4534,Z 168,A -12.4992,B 9.9693,C 0.2729,E1 10.1281,E2 463.839} C_DIS
LIN {X 135.0103,Y -36.6198,Z 168,A -13.957,B 9.9697,C 0.2609,E1 10.1272,E2 465.2065} C_DIS
LIN {X 134.3081,Y -39.1128,Z 168,A -15.144,B 9.9695,C 0.2671,E1 10.1262,E2 466.4109} C_DIS
LIN {X 133.1349,Y -42.938,Z 168,A -16.6971,B 9.9695,C 0.2696,E1 10.1249,E2 467.9547} C_DIS
LIN {X 131.7024,Y -47.1486,Z 168,A -18.6264,B 9.9692,C 0.2774,E1 10.1231,E2 469.8998} C_DIS
LIN {X 130.1476,Y -51.2876,Z 168,A -20.3295,B 9.9692,C 0.2797,E1 10.1214,E2 471.5911} C_DIS
LIN {X 128.7044,Y -54.8102,Z 168,A -21.7607,B 9.9692,C 0.2807,E1 10.1199,E2 473.0075} C_DIS
LIN {X 127.5006,Y -57.552,Z 168,A -22.9861,B 9.969,C 0.284,E1 10.1185,E2 474.234} C_DIS
LIN {X 126.1072,Y -60.5428,Z 168,A -24.281,B 9.969,C 0.2862,E1 10.117,E2 475.5231} C_DIS
LIN {X 124.0271,Y -64.6977,Z 168,A -26.0425,B 9.969,C 0.2877,E1 10.1148,E2 477.2684} C_DIS
LIN {X 122.6446,Y -67.2857,Z 168,A -27.4716,B 9.9687,C 0.2966,E1 10.1128,E2 478.7282} C_DIS
LIN {X 120.5956,Y -70.8917,Z 168,A -29.395,B 9.9684,C 0.3066,E1 10.1101,E2 480.6824} C_DIS
LIN {X 118.7856,Y -73.8845,Z 168,A -30.5846,B 9.9684,C 0.3041,E1 10.1084,E2 481.8423} C_DIS
LIN {X 116.2461,Y -77.8191,Z 168,A -32.9166,B 9.968,C 0.3192,E1 10.1047,E2 484.2296} C_DIS
LIN {X 113.5563,Y -81.695,Z 168,A -34.3091,B 9.9682,C 0.3105,E1 10.1026,E2 485.5547} C_DIS
LIN {X 111.2627,Y -84.7915,Z 168,A -35.9486,B 9.9681,C 0.3159,E1 10.0998,E2 487.2038} C_DIS
LIN {X 108.6087,Y -88.1661,Z 168,A -37.6631,B 9.968,C 0.3189,E1 10.0968,E2 488.9146} C_DIS
LIN {X 105.7879,Y -91.5312,Z 168,A -39.3196,B 9.968,C 0.3195,E1 10.0939,E2 490.5546} C_DIS
LIN {X 101.7145,Y -96.037,Z 168,A -41.8709,B 9.9677,C 0.3266,E1 10.0891,E2 493.1168} C_DIS
LIN {X 98.8,Y -99.0333,Z 168,A -43.72,B 9.9675,C 0.3337,E1 10.0854,E2 494.9854} C_DIS
LIN {X 95.0247,Y -102.6617,Z 168,A -46.0654,B 9.9672,C 0.3431,E1 10.0805,E2 497.3589} C_DIS
LIN {X 92.0262,Y -105.3571,Z 168,A -47.2366,B 9.9675,C 0.3347,E1 10.0782,E2 498.4696} C_DIS
LIN {X 89.0312,Y -107.9001,Z 168,A -49.0416,B 9.9672,C 0.3426,E1 10.0743,E2 500.3016} C_DIS
LIN {X 85.333,Y -110.8486,Z 168,A -51.4095,B 9.9667,C 0.3567,E1 10.0689,E2 502.7269} C_DIS
LIN {X 81.2004,Y -113.91,Z 168,A -52.9515,B 9.9671,C 0.3469,E1 10.0656,E2 504.1982} C_DIS
LIN {X 77.8225,Y -116.2439,Z 168,A -54.6061,B 9.967,C 0.3492,E1 10.0618,E2 505.8509} C_DIS
LIN {X 73.6349,Y -118.941,Z 168,A -56.647,B 9.9669,C 0.3526,E1 10.057,E2 507.8938} C_DIS
LIN {X 70.2018,Y -120.9987,Z 168,A -58.2836,B 9.9668,C 0.3551,E1 10.053,E2 509.5315} C_DIS
LIN {X 66.4106,Y -123.1204,Z 168,A -60.0398,B 9.9667,C 0.3572,E1 10.0487,E2 511.2862} C_DIS
LIN {X 63.144,Y -124.8252,Z 168,A -61.4834,B 9.9667,C 0.3578,E1 10.0452,E2 512.7226} C_DIS
LIN {X 58.5414,Y -127.0485,Z 168,A -63.5636,B 9.9666,C 0.3604,E1 10.0399,E2 514.8029} C_DIS
LIN {X 55.0272,Y -128.6106,Z 168,A -65.174,B 9.9665,C 0.3632,E1 10.0358,E2 516.4192} C_DIS
LIN {X 49.9781,Y -130.6567,Z 168,A -67.5794,B 9.9662,C 0.37,E1 10.0295,E2 518.849} C_DIS
LIN {X 45.7967,Y -132.1782,Z 168,A -69.1567,B 9.9664,C 0.3662,E1 10.0254,E2 520.3959} C_DIS
LIN {X 42.1047,Y -133.4011,Z 168,A -70.6889,B 9.9664,C 0.3664,E1 10.0213,E2 521.9214} C_DIS
LIN {X 39.2833,Y -134.2582,Z 168,A -71.9484,B 9.9663,C 0.3688,E1 10.018,E2 523.1885} C_DIS
LIN {X 35.6993,Y -135.2558,Z 168,A -73.4426,B 9.9663,C 0.3694,E1 10.0139,E2 524.68} C_DIS
LIN {X 32.4436,Y -136.0735,Z 168,A -75.1134,B 9.966,C 0.3774,E1 10.0093,E2 526.39} C_DIS
LIN {X 29.0615,Y -136.8361,Z 168,A -76.2069,B 9.9662,C 0.3709,E1 10.0064,E2 527.4423} C_DIS
LIN {X 26.0003,Y -137.4501,Z 168,A -77.4907,B 9.9662,C 0.3719,E1 10.0029,E2 528.7276} C_DIS
LIN {X 22.7064,Y -138.0326,Z 168,A -78.8424,B 9.9662,C 0.3723,E1 9.9992,E2 530.0777} C_DIS
LIN {X 19.1423,Y -138.5731,Z 168,A -80.4164,B 9.966,C 0.3754,E1 9.9948,E2 531.6653} C_DIS
LIN {X 15.03,Y -139.0777,Z 168,A -82.3162,B 9.9658,C 0.3808,E1 9.9894,E2 533.5922} C_DIS
LIN {X 11.706,Y -139.3969,Z 168,A -83.3982,B 9.9661,C 0.3748,E1 9.9865,E2 534.6381} C_DIS
LIN {X 8.5784,Y -139.6243,Z 168,A -84.7262,B 9.9661,C 0.3762,E1 9.9828,E2 535.9725} C_DIS
LIN {X 5.1043,Y -139.7949,Z 168,A -86.049,B 9.9661,C 0.3742,E1 9.9792,E2 537.2828} C_DIS
LIN {X 2.3281,Y -139.8683,Z 168,A -87.2392,B 9.9661,C 0.3756,E1 9.9758,E2 538.4804} C_DIS
LIN {X 2.3281,Y -139.8683,Z 168,A -87.2392,B 9.9661,C 0.3756,E1 9.9758,E2 538.4804} C_DIS
Enddeposition()
LIN {X 1.0098,Y -140.7961,Z 168,A -87.2825,B 9.9664,C 0.3704,E1 9.9759,E2 538.4933} C_DIS
Startdeposition()
$VEL.CP = VEL_PRINT
LIN {X 4.0961,Y -140.7421,Z 168,A -85.8852,B 9.9664,C 0.3669,E1 9.9799,E2 537.0768} C_DIS
LIN {X 8.1005,Y -140.5694,Z 168,A -84.1118,B 9.9666,C 0.3632,E1 9.9849,E2 535.2838} C_DIS
LIN {X 12.6203,Y -140.2369,Z 168,A -82.231,B 9.9666,C 0.3617,E1 9.9901,E2 533.3972} C_DIS
LIN {X 17.2466,Y -139.7424,Z 168,A -80.4001,B 9.9666,C 0.3623,E1 9.9952,E2 531.5734} C_DIS
LIN {X 20.6628,Y -139.2791,Z 168,A -79.0769,B 9.9666,C 0.3634,E1 9.9988,E2 530.26} C_DIS
LIN {X 24.4061,Y -138.6706,Z 168,A -77.5214,B 9.9666,C 0.3621,E1 10.0031,E2 528.7018} C_DIS
LIN {X 27.9827,Y -137.9927,Z 168,A -76.2383,B 9.9666,C 0.3658,E1 10.0066,E2 527.4438} C_DIS
LIN {X 30.8304,Y -137.3855,Z 168,A -74.9075,B 9.9666,C 0.3615,E1 10.0102,E2 526.0931} C_DIS
LIN {X 34.2116,Y -136.5824,Z 168,A -73.4975,B 9.9667,C 0.3604,E1 10.0141,E2 524.6826} C_DIS
LIN {X 38.0753,Y -135.5555,Z 168,A -71.8849,B 9.9667,C 0.3593,E1 10.0184,E2 523.0707} C_DIS
LIN {X 41.3884,Y -134.5809,Z 168,A -70.4194,B 9.9669,C 0.3565,E1 10.0224,E2 521.5962} C_DIS
LIN {X 45.8061,Y -133.1423,Z 168,A -68.6055,B 9.9669,C 0.3564,E1 10.0271,E2 519.791} C_DIS
LIN {X 48.6699,Y -132.1241,Z 168,A -67.2855,B 9.9669,C 0.353,E1 10.0306,E2 518.4591} C_DIS
LIN {X 52.374,Y -130.6981,Z 168,A -65.781,B 9.9669,C 0.3537,E1 10.0345,E2 516.9679} C_DIS
LIN {X 55.96,Y -129.2031,Z 168,A -64.1527,B 9.9671,C 0.3506,E1 10.0387,E2 515.3319} C_DIS
LIN {X 59.674,Y -127.5318,Z 168,A -62.4404,B 9.9672,C 0.3471,E1 10.0431,E2 513.6111} C_DIS
LIN {X 63.3166,Y -125.763,Z 168,A -60.849,B 9.9672,C 0.3461,E1 10.047,E2 512.0257} C_DIS
LIN {X 66.6141,Y -124.0486,Z 168,A -59.321,B 9.9673,C 0.3435,E1 10.0508,E2 510.4943} C_DIS
LIN {X 70.3834,Y -121.9496,Z 168,A -57.5741,B 9.9674,C 0.341,E1 10.0551,E2 508.7469} C_DIS
LIN {X 74.3658,Y -119.5626,Z 168,A -55.7061,B 9.9674,C 0.3385,E1 10.0595,E2 506.8801} C_DIS
LIN {X 78.2286,Y -117.0717,Z 168,A -53.8473,B 9.9676,C 0.3356,E1 10.0639,E2 505.021} C_DIS
LIN {X 82.0131,Y -114.4525,Z 168,A -51.987,B 9.9676,C 0.3325,E1 10.0681,E2 503.1607} C_DIS
LIN {X 85.827,Y -111.6215,Z 168,A -50.1525,B 9.9677,C 0.3314,E1 10.0722,E2 501.3373} C_DIS
LIN {X 88.8647,Y -109.2183,Z 168,A -48.5035,B 9.9679,C 0.3266,E1 10.0758,E2 499.6771} C_DIS
LIN {X 92.3024,Y -106.3291,Z 168,A -46.6745,B 9.968,C 0.3229,E1 10.0797,E2 497.8461} C_DIS
LIN {X 95.8349,Y -103.1561,Z 168,A -44.7933,B 9.968,C 0.3202,E1 10.0835,E2 495.9696} C_DIS
LIN {X 98.9526,Y -100.1701,Z 168,A -43.097,B 9.9682,C 0.318,E1 10.0869,E2 494.2795} C_DIS
LIN {X 101.9765,Y -97.0894,Z 168,A -41.2992,B 9.9683,C 0.3131,E1 10.0904,E2 492.4744} C_DIS
LIN {X 104.926,Y -93.8937,Z 168,A -39.5762,B 9.9684,C 0.3103,E1 10.0936,E2 490.7557} C_DIS
LIN {X 107.9128,Y -90.4451,Z 168,A -37.7344,B 9.9685,C 0.3064,E1 10.097,E2 488.9139} C_DIS
LIN {X 110.8371,Y -86.8369,Z 168,A -35.874,B 9.9686,C 0.3027,E1 10.1002,E2 487.0553} C_DIS
LIN {X 113.6043,Y -83.1842,Z 168,A -34.0105,B 9.9688,C 0.2983,E1 10.1033,E2 485.1901} C_DIS
LIN {X 116.2624,Y -79.4269,Z 168,A -32.1612,B 9.9688,C 0.2943,E1 10.1063,E2 483.3418} C_DIS
LIN {X 118.8149,Y -75.5559,Z 168,A -30.3015,B 9.969,C 0.2902,E1 10.1091,E2 481.4837} C_DIS
LIN {X 121.2145,Y -71.6428,Z 168,A -28.5083,B 9.969,C 0.2874,E1 10.1117,E2 479.6983} C_DIS
LIN {X 123.3542,Y -67.8924,Z 168,A -26.7738,B 9.9692,C 0.2834,E1 10.114,E2 477.9649} C_DIS
LIN {X 125.1105,Y -64.5983,Z 168,A -25.3416,B 9.9692,C 0.2816,E1 10.1159,E2 476.5425} C_DIS
LIN {X 126.9165,Y -60.969,Z 168,A -23.6508,B 9.9694,C 0.2761,E1 10.118,E2 474.8444} C_DIS
LIN {X 128.3724,Y -57.8414,Z 168,A -22.2508,B 9.9694,C 0.2724,E1 10.1196,E2 473.4433} C_DIS
LIN {X 130.0835,Y -53.8832,Z 168,A -20.5358,B 9.9696,C 0.2687,E1 10.1214,E2 471.7316} C_DIS
LIN {X 131.5596,Y -50.1771,Z 168,A -18.9901,B 9.9696,C 0.2662,E1 10.123,E2 470.1945} C_DIS
LIN {X 132.7521,Y -46.9315,Z 168,A -17.4346,B 9.9699,C 0.2584,E1 10.1245,E2 468.6179} C_DIS
LIN {X 133.8642,Y -43.6585,Z 168,A -16.2196,B 9.9699,C 0.2594,E1 10.1255,E2 467.4266} C_DIS
LIN {X 134.739,Y -40.8719,Z 168,A -15.0443,B 9.9699,C 0.2564,E1 10.1265,E2 466.2517} C_DIS
LIN {X 135.7007,Y -37.5558,Z 168,A -13.5875,B 9.9701,C 0.2511,E1 10.1276,E2 464.7866} C_DIS
LIN {X 136.7184,Y -33.6682,Z 168,A -12.1066,B 9.9701,C 0.2504,E1 10.1286,E2 463.3242} C_DIS
LIN {X 137.4992,Y -30.3211,Z 168,A -10.7533,B 9.9701,C 0.2476,E1 10.1295,E2 461.9754} C_DIS
LIN {X 138.1006,Y -27.4527,Z 168,A -9.5008,B 9.9703,C 0.2426,E1 10.1302,E2 460.7137} C_DIS
LIN {X 138.8208,Y -23.536,Z 168,A -7.8907,B 9.9703,C 0.2382,E1 10.1309,E2 459.1033} C_DIS
LIN {X 139.2804,Y -20.6535,Z 168,A -6.7128,B 9.9704,C 0.235,E1 10.1314,E2 457.9255} C_DIS
LIN {X 139.8071,Y -16.7037,Z 168,A -5.1283,B 9.9705,C 0.2312,E1 10.132,E2 456.3441} C_DIS
LIN {X 140.2378,Y -12.6092,Z 168,A -3.3356,B 9.9707,C 0.2233,E1 10.1325,E2 454.5344} C_DIS
LIN {X 140.5697,Y -8.0962,Z 168,A -1.5263,B 9.9708,C 0.2187,E1 10.1328,E2 452.7274} C_DIS
LIN {X 140.76,Y -3.4538,Z 168,A 0.1832,B 9.9708,C 0.2179,E1 10.133,E2 451.0397} C_DIS
LIN {X 140.8059,Y -0.001,Z 168,A 1.7747,B 9.971,C 0.209,E1 10.133,E2 449.4225} C_DIS
LIN {X 140.745,Y 3.9914,Z 168,A 3.2049,B 9.971,C 0.2092,E1 10.1329,E2 448.0161} C_DIS
LIN {X 140.5692,Y 8.1039,Z 168,A 4.991,B 9.9712,C 0.2015,E1 10.1326,E2 446.2139} C_DIS
LIN {X 140.2375,Y 12.6133,Z 168,A 6.8152,B 9.9712,C 0.1966,E1 10.1322,E2 444.3901} C_DIS
LIN {X 139.7405,Y 17.2627,Z 168,A 8.6319,B 9.9713,C 0.1933,E1 10.1316,E2 442.5829} C_DIS
LIN {X 139.2772,Y 20.6756,Z 168,A 9.9005,B 9.9713,C 0.1927,E1 10.1311,E2 441.3303} C_DIS
LIN {X 138.6354,Y 24.6028,Z 168,A 11.5048,B 9.9714,C 0.1884,E1 10.1304,E2 439.7265} C_DIS
LIN {X 137.9917,Y 27.9878,Z 168,A 12.7412,B 9.9714,C 0.1886,E1 10.1297,E2 438.5104} C_DIS
LIN {X 137.3851,Y 30.8323,Z 168,A 14.091,B 9.9716,C 0.181,E1 10.1289,E2 437.138} C_DIS
LIN {X 136.5824,Y 34.2116,Z 168,A 15.4477,B 9.9716,C 0.1785,E1 10.128,E2 435.7875} C_DIS
LIN {X 135.4858,Y 38.3245,Z 168,A 17.243,B 9.9717,C 0.172,E1 10.1267,E2 433.9825} C_DIS
LIN {X 134.2259,Y 42.5265,Z 168,A 18.9131,B 9.9717,C 0.17,E1 10.1253,E2 432.3259} C_DIS
LIN {X 133.1428,Y 45.8048,Z 168,A 20.298,B 9.9718,C 0.1666,E1 10.1241,E2 430.9425} C_DIS
LIN {X 131.9651,Y 49.0943,Z 168,A 21.699,B 9.9718,C 0.1633,E1 10.1227,E2 429.5432} C_DIS
LIN {X 130.7244,Y 52.3089,Z 168,A 23.0807,B 9.9719,C 0.16,E1 10.1213,E2 428.163} C_DIS
LIN {X 129.1971,Y 55.9739,Z 168,A 24.723,B 9.9719,C 0.1551,E1 10.1195,E2 426.5162} C_DIS
LIN {X 127.5401,Y 59.656,Z 168,A 26.4098,B 9.9721,C 0.1496,E1 10.1176,E2 424.8226} C_DIS
LIN {X 125.7672,Y 63.3083,Z 168,A 27.9977,B 9.9721,C 0.147,E1 10.1156,E2 423.2418} C_DIS
LIN {X 124.051,Y 66.6096,Z 168,A 29.5269,B 9.9721,C 0.1427,E1 10.1136,E2 421.7098} C_DIS
LIN {X 121.9356,Y 70.4075,Z 168,A 31.2676,B 9.9722,C 0.139,E1 10.1112,E2 419.9716} C_DIS
LIN {X 119.553,Y 74.3813,Z 168,A 33.0765,B 9.9722,C 0.1363,E1 10.1086,E2 418.1716} C_DIS
LIN {X 117.3547,Y 77.8047,Z 168,A 34.7749,B 9.9723,C 0.1312,E1 10.106,E2 416.4667} C_DIS
LIN {X 114.9632,Y 81.2956,Z 168,A 36.4741,B 9.9723,C 0.1277,E1 10.1033,E2 414.7694} C_DIS
LIN {X 112.2141,Y 85.0504,Z 168,A 38.3408,B 9.9724,C 0.124,E1 10.1001,E2 412.9053} C_DIS
LIN {X 109.3885,Y 88.6553,Z 168,A 40.1979,B 9.9724,C 0.12,E1 10.0969,E2 411.0482} C_DIS
LIN {X 106.4427,Y 92.1715,Z 168,A 41.9378,B 9.9724,C 0.119,E1 10.0938,E2 409.3237} C_DIS
LIN {X 103.7384,Y 95.2043,Z 168,A 43.6136,B 9.9725,C 0.115,E1 10.0906,E2 407.6444} C_DIS
LIN {X 100.7748,Y 98.3364,Z 168,A 45.3929,B 9.9725,C 0.1107,E1 10.0872,E2 405.8612} C_DIS
LIN {X 97.7161,Y 101.3763,Z 168,A 47.1532,B 9.9726,C 0.1071,E1 10.0837,E2 404.0997} C_DIS
LIN {X 94.5562,Y 104.3294,Z 168,A 48.8802,B 9.9726,C 0.1045,E1 10.0801,E2 402.3763} C_DIS
LIN {X 91.1036,Y 107.3575,Z 168,A 50.7333,B 9.9726,C 0.1013,E1 10.0762,E2 400.5246} C_DIS
LIN {X 87.771,Y 110.0989,Z 168,A 52.4678,B 9.9726,C 0.0987,E1 10.0725,E2 398.7925} C_DIS
LIN {X 85.0443,Y 112.2187,Z 168,A 53.808,B 9.9727,C 0.0978,E1 10.0695,E2 397.4604} C_DIS
LIN {X 81.6761,Y 114.6934,Z 168,A 55.5495,B 9.9727,C 0.094,E1 10.0655,E2 395.7133} C_DIS
LIN {X 78.2297,Y 117.0709,Z 168,A 57.1905,B 9.9727,C 0.0928,E1 10.0618,E2 394.08} C_DIS
LIN {X 74.8209,Y 119.279,Z 168,A 58.8352,B 9.9727,C 0.0904,E1 10.0579,E2 392.4362} C_DIS
LIN {X 71.4117,Y 121.3502,Z 168,A 60.4868,B 9.9728,C 0.0874,E1 10.0539,E2 390.7807} C_DIS
LIN {X 67.79,Y 123.4106,Z 168,A 62.1714,B 9.9728,C 0.0853,E1 10.0498,E2 389.0974} C_DIS
LIN {X 64.3998,Y 125.2116,Z 168,A 63.6531,B 9.9728,C 0.0852,E1 10.0462,E2 387.6259} C_DIS
LIN {X 61.4008,Y 126.7102,Z 168,A 65.1101,B 9.9728,C 0.0813,E1 10.0425,E2 386.1571} C_DIS
LIN {X 57.8361,Y 128.3747,Z 168,A 66.6451,B 9.9728,C 0.0809,E1 10.0386,E2 384.6304} C_DIS
LIN {X 53.8755,Y 130.0867,Z 168,A 68.3756,B 9.9728,C 0.0796,E1 10.0342,E2 382.9033} C_DIS
LIN {X 50.0957,Y 131.5901,Z 168,A 69.9365,B 9.9728,C 0.0801,E1 10.0301,E2 381.3546} C_DIS
LIN {X 46.9317,Y 132.752,Z 168,A 71.5017,B 9.9729,C 0.0743,E1 10.026,E2 379.7648} C_DIS
LIN {X 43.6587,Y 133.8641,Z 168,A 72.9029,B 9.9729,C 0.0732,E1 10.0223,E2 378.3646} C_DIS
LIN {X 39.6709,Y 135.0971,Z 168,A 74.5089,B 9.9729,C 0.074,E1 10.018,E2 376.7706} C_DIS
LIN {X 35.3378,Y 136.2966,Z 168,A 76.2518,B 9.9729,C 0.0746,E1 10.0133,E2 375.0392} C_DIS
LIN {X 32.4828,Y 137.0042,Z 168,A 77.5205,B 9.9729,C 0.0722,E1 10.0098,E2 373.7615} C_DIS
LIN {X 28.9234,Y 137.8009,Z 168,A 78.9095,B 9.9729,C 0.0735,E1 10.0061,E2 372.3851} C_DIS
LIN {X 25.7554,Y 138.4275,Z 168,A 80.3535,B 9.9729,C 0.0699,E1 10.0021,E2 370.9248} C_DIS
LIN {X 21.8302,Y 139.0991,Z 168,A 81.6812,B 9.9729,C 0.0758,E1 9.9985,E2 369.6348} C_DIS
LIN {X 18.9433,Y 139.5228,Z 168,A 83.1624,B 9.9729,C 0.0688,E1 9.9943,E2 368.1166} C_DIS
LIN {X 14.8139,Y 140.0202,Z 168,A 84.7686,B 9.9729,C 0.0702,E1 9.9899,E2 366.522} C_DIS
LIN {X 10.3442,Y 140.4211,Z 168,A 86.6173,B 9.9729,C 0.0693,E1 9.9848,E2 364.6711} C_DIS
LIN {X 5.7132,Y 140.6858,Z 168,A 88.5174,B 9.9729,C 0.0688,E1 9.9794,E2 362.7703} C_DIS
LIN {X 1.7281,Y 140.7924,Z 168,A 90.1806,B 9.9729,C 0.0679,E1 9.9748,E2 361.1026} C_DIS
LIN {X -2.2744,Y 140.7833,Z 168,A 91.6856,B 9.9729,C 0.0707,E1 9.9706,E2 359.614} C_DIS
LIN {X -5.7246,Y 140.6854,Z 168,A 93.191,B 9.9729,C 0.0687,E1 9.9664,E2 358.0964} C_DIS
LIN {X -10.3608,Y 140.4198,Z 168,A 95.035,B 9.9729,C 0.0701,E1 9.9613,E2 356.2592} C_DIS
LIN {X -15.0284,Y 139.9972,Z 168,A 96.9621,B 9.9729,C 0.0703,E1 9.9559,E2 354.3307} C_DIS
LIN {X -19.5045,Y 139.4446,Z 168,A 98.5713,B 9.9729,C 0.076,E1 9.9515,E2 352.7513} C_DIS
LIN {X -22.3832,Y 139.0132,Z 168,A 100.0628,B 9.9729,C 0.0699,E1 9.9473,E2 351.2215} C_DIS
LIN {X -26.2878,Y 138.3257,Z 168,A 101.5813,B 9.9729,C 0.0729,E1 9.9432,E2 349.7161} C_DIS
LIN {X -30.3299,Y 137.4973,Z 168,A 103.3343,B 9.9729,C 0.0724,E1 9.9384,E2 347.9548} C_DIS
LIN {X -34.2136,Y 136.5819,Z 168,A 104.8553,B 9.9729,C 0.0757,E1 9.9343,E2 346.4479} C_DIS
LIN {X -38.0724,Y 135.5563,Z 168,A 106.4846,B 9.9729,C 0.0769,E1 9.9299,E2 344.8192} C_DIS
LIN {X -41.3932,Y 134.5794,Z 168,A 107.9658,B 9.9729,C 0.0766,E1 9.9259,E2 343.3298} C_DIS
LIN {X -45.8113,Y 133.1405,Z 168,A 109.7984,B 9.9729,C 0.0797,E1 9.9211,E2 341.506} C_DIS
LIN {X -49.0595,Y 131.9782,Z 168,A 111.2088,B 9.9729,C 0.081,E1 9.9174,E2 340.0958} C_DIS
LIN {X -52.2782,Y 130.7367,Z 168,A 112.6199,B 9.9729,C 0.0824,E1 9.9137,E2 338.6849} C_DIS
LIN {X -55.9589,Y 129.2035,Z 168,A 114.2045,B 9.9729,C 0.0851,E1 9.9097,E2 337.1064} C_DIS
LIN {X -58.6366,Y 128.0115,Z 168,A 115.5198,B 9.9729,C 0.084,E1 9.9063,E2 335.7765} C_DIS
LIN {X -61.8021,Y 126.5137,Z 168,A 116.8829,B 9.9729,C 0.0872,E1 9.9029,E2 334.4225} C_DIS
LIN {X -65.1183,Y 124.8386,Z 168,A 118.3639,B 9.9728,C 0.0899,E1 9.8992,E2 332.9467} C_DIS
LIN {X -68.6639,Y 122.9264,Z 168,A 120.1206,B 9.9728,C 0.0899,E1 9.8949,E2 331.1766} C_DIS
LIN {X -72.3849,Y 120.7727,Z 168,A 121.8335,B 9.9728,C 0.0932,E1 9.8908,E2 329.4699} C_DIS
LIN {X -75.5636,Y 118.81,Z 168,A 123.4809,B 9.9728,C 0.093,E1 9.8868,E2 327.8077} C_DIS
LIN {X -79.4407,Y 116.2529,Z 168,A 125.3669,B 9.9728,C 0.0963,E1 9.8825,E2 325.924} C_DIS
LIN {X -83.1805,Y 113.607,Z 168,A 127.2526,B 9.9727,C 0.0991,E1 9.8782,E2 324.0373} C_DIS
LIN {X -86.844,Y 110.8315,Z 168,A 129.136,B 9.9727,C 0.1022,E1 9.874,E2 322.154} C_DIS
LIN {X -90.4519,Y 107.9071,Z 168,A 131.029,B 9.9727,C 0.1057,E1 9.8699,E2 320.2625} C_DIS
LIN {X -93.9151,Y 104.9069,Z 168,A 132.8732,B 9.9726,C 0.1098,E1 9.8661,E2 318.4227} C_DIS
LIN {X -97.0976,Y 101.9687,Z 168,A 134.7162,B 9.9726,C 0.1118,E1 9.8623,E2 316.5712} C_DIS
LIN {X -100.176,Y 98.9466,Z 168,A 136.4364,B 9.9726,C 0.1161,E1 9.8589,E2 314.8573} C_DIS
LIN {X -103.16,Y 95.8307,Z 168,A 138.2636,B 9.9725,C 0.1185,E1 9.8554,E2 313.0228} C_DIS
LIN {X -106.068,Y 92.6017,Z 168,A 139.9919,B 9.9725,C 0.1232,E1 9.8522,E2 311.3014} C_DIS
LIN {X -108.8517,Y 89.3133,Z 168,A 141.8159,B 9.9724,C 0.1258,E1 9.849,E2 309.4703} C_DIS
LIN {X -111.5322,Y 85.9432,Z 168,A 143.5455,B 9.9724,C 0.1303,E1 9.846,E2 307.7454} C_DIS
LIN {X -114.1073,Y 82.4927,Z 168,A 145.3907,B 9.9724,C 0.1327,E1 9.8429,E2 305.8901} C_DIS
LIN {X -116.7415,Y 78.7208,Z 168,A 147.2139,B 9.9722,C 0.1382,E1 9.8401,E2 304.0752} C_DIS
LIN {X -118.9624,Y 75.3225,Z 168,A 148.8882,B 9.9722,C 0.1419,E1 9.8375,E2 302.3998} C_DIS
LIN {X -121.2155,Y 71.6411,Z 168,A 150.6743,B 9.9722,C 0.1457,E1 9.835,E2 300.6118} C_DIS
LIN {X -123.3546,Y 67.8917,Z 168,A 152.455,B 9.9721,C 0.1498,E1 9.8325,E2 298.83} C_DIS
LIN {X -125.1339,Y 64.5523,Z 168,A 153.947,B 9.972,C 0.1547,E1 9.8306,E2 297.3457} C_DIS
LIN {X -126.8313,Y 61.1474,Z 168,A 155.5931,B 9.972,C 0.1569,E1 9.8286,E2 295.6887} C_DIS
LIN {X -128.4009,Y 57.7776,Z 168,A 157.1197,B 9.972,C 0.1607,E1 9.8268,E2 294.162} C_DIS
LIN {X -130.0819,Y 53.8869,Z 168,A 158.866,B 9.9718,C 0.165,E1 9.8249,E2 292.4147} C_DIS
LIN {X -131.5611,Y 50.1732,Z 168,A 160.4562,B 9.9718,C 0.1701,E1 9.8233,E2 290.831} C_DIS
LIN {X -132.752,Y 46.9317,Z 168,A 162.0572,B 9.9718,C 0.1703,E1 9.8218,E2 289.2065} C_DIS
LIN {X -133.8643,Y 43.6581,Z 168,A 163.4835,B 9.9717,C 0.1738,E1 9.8205,E2 287.7793} C_DIS
LIN {X -135.2297,Y 39.2179,Z 168,A 165.2271,B 9.9715,C 0.1819,E1 9.8191,E2 286.0564} C_DIS
LIN {X -136.2882,Y 35.3708,Z 168,A 166.8834,B 9.9715,C 0.1859,E1 9.8179,E2 284.3978} C_DIS
LIN {X -137.2623,Y 31.3697,Z 168,A 168.3886,B 9.9713,C 0.194,E1 9.817,E2 282.9161} C_DIS
LIN {X -137.7939,Y 28.9561,Z 168,A 169.7149,B 9.9713,C 0.1907,E1 9.8162,E2 281.5499} C_DIS
LIN {X -138.5575,Y 25.0379,Z 168,A 171.2079,B 9.9713,C 0.1979,E1 9.8154,E2 280.0754} C_DIS
LIN {X -139.0973,Y 21.8416,Z 168,A 172.4142,B 9.9711,C 0.2039,E1 9.8149,E2 278.8849} C_DIS
LIN {X -139.5214,Y 18.954,Z 168,A 173.9324,B 9.9711,C 0.201,E1 9.8143,E2 277.3256} C_DIS
LIN {X -140.0614,Y 14.4317,Z 168,A 175.6767,B 9.9711,C 0.2085,E1 9.8137,E2 275.5972} C_DIS
LIN {X -140.423,Y 10.3176,Z 168,A 177.4452,B 9.971,C 0.2117,E1 9.8133,E2 273.8191} C_DIS
LIN {X -140.6861,Y 5.7069,Z 168,A 179.3698,B 9.9709,C 0.2163,E1 9.8131,E2 271.8905} C_DIS
LIN {X -140.7929,Y 1.6956,Z 168,A -179.143,B 9.9707,C 0.2239,E1 9.813,E2 270.4238} C_DIS
LIN {X -140.7833,Y -2.2722,Z 168,A -177.3898,B 9.9707,C 0.2259,E1 9.813,E2 268.6543} C_DIS
LIN {X -140.6823,Y -5.8029,Z 168,A -175.8517,B 9.9706,C 0.2282,E1 9.8132,E2 267.1046} C_DIS
LIN {X -140.4172,Y -10.3975,Z 168,A -174.0729,B 9.9704,C 0.2354,E1 9.8135,E2 265.3396} C_DIS
LIN {X -140.1238,Y -13.8024,Z 168,A -172.6532,B 9.9704,C 0.2389,E1 9.8139,E2 263.9175} C_DIS
LIN {X -139.6771,Y -17.7663,Z 168,A -170.9868,B 9.9703,C 0.2428,E1 9.8144,E2 262.2471} C_DIS
LIN {X -139.2796,Y -20.6588,Z 168,A -169.8007,B 9.9702,C 0.2462,E1 9.8149,E2 261.0623} C_DIS
LIN {X -138.6889,Y -24.3036,Z 168,A -168.1885,B 9.9702,C 0.2484,E1 9.8157,E2 259.4374} C_DIS
LIN {X -137.9903,Y -27.9948,Z 168,A -166.8597,B 9.9699,C 0.2566,E1 9.8164,E2 258.1356} C_DIS
LIN {X -137.3811,Y -30.8497,Z 168,A -165.5046,B 9.9699,C 0.2567,E1 9.8172,E2 256.76} C_DIS
LIN {X -136.5829,Y -34.2096,Z 168,A -164.0789,B 9.9699,C 0.2603,E1 9.8181,E2 255.3328} C_DIS
LIN {X -135.5553,Y -38.0758,Z 168,A -162.4325,B 9.9697,C 0.2645,E1 9.8193,E2 253.6854} C_DIS
LIN {X -134.5812,Y -41.3875,Z 168,A -160.9389,B 9.9697,C 0.2666,E1 9.8205,E2 252.1814} C_DIS
LIN {X -133.1044,Y -45.9154,Z 168,A -159.0715,B 9.9695,C 0.2733,E1 9.8222,E2 250.3247} C_DIS
LIN {X -131.9817,Y -49.0501,Z 168,A -157.6687,B 9.9694,C 0.2761,E1 9.8235,E2 248.9168} C_DIS
LIN {X -130.7402,Y -52.2697,Z 168,A -156.2418,B 9.9694,C 0.2794,E1 9.825,E2 247.4879} C_DIS
LIN {X -129.1289,Y -56.1314,Z 168,A -154.4965,B 9.9692,C 0.283,E1 9.8269,E2 245.7384} C_DIS
LIN {X -127.536,Y -59.6649,Z 168,A -152.806,B 9.9692,C 0.2849,E1 9.8289,E2 244.0343} C_DIS
LIN {X -125.7678,Y -63.3071,Z 168,A -151.1794,B 9.969,C 0.2896,E1 9.8309,E2 242.4115} C_DIS
LIN {X -124.0519,Y -66.6079,Z 168,A -149.6187,B 9.969,C 0.2925,E1 9.833,E2 240.8457} C_DIS
LIN {X -121.9519,Y -70.3794,Z 168,A -147.8337,B 9.9688,C 0.2963,E1 9.8354,E2 239.0581} C_DIS
LIN {X -119.5061,Y -74.4566,Z 168,A -145.9478,B 9.9687,C 0.302,E1 9.8382,E2 237.1797} C_DIS
LIN {X -117.4024,Y -77.7323,Z 168,A -144.2537,B 9.9687,C 0.3036,E1 9.8408,E2 235.4722} C_DIS
LIN {X -114.9639,Y -81.2946,Z 168,A -142.4827,B 9.9685,C 0.3074,E1 9.8436,E2 233.7003} C_DIS
LIN {X -112.212,Y -85.0531,Z 168,A -140.5769,B 9.9684,C 0.3115,E1 9.8468,E2 231.7941} C_DIS
LIN {X -109.3881,Y -88.6558,Z 168,A -138.654,B 9.9683,C 0.3144,E1 9.8501,E2 229.8643} C_DIS
LIN {X -106.4285,Y -92.188,Z 168,A -136.7756,B 9.9682,C 0.3184,E1 9.8535,E2 227.9863} C_DIS
LIN {X -103.5564,Y -95.4022,Z 168,A -135.02,B 9.968,C 0.322,E1 9.8568,E2 226.2312} C_DIS
LIN {X -100.363,Y -98.7563,Z 168,A -133.1798,B 9.9679,C 0.3267,E1 9.8604,E2 224.3976} C_DIS
LIN {X -97.5193,Y -101.5656,Z 168,A -131.4619,B 9.9679,C 0.328,E1 9.8639,E2 222.6683} C_DIS
LIN {X -94.0993,Y -104.7419,Z 168,A -129.6069,B 9.9677,C 0.3325,E1 9.8677,E2 220.8196} C_DIS
LIN {X -91.1069,Y -107.3547,Z 168,A -127.9236,B 9.9677,C 0.334,E1 9.8713,E2 219.1281} C_DIS
LIN {X -87.7722,Y -110.0979,Z 168,A -126.1569,B 9.9675,C 0.3369,E1 9.8751,E2 217.3606} C_DIS
LIN {X -84.3562,Y -112.737,Z 168,A -124.3679,B 9.9675,C 0.3392,E1 9.8791,E2 215.5677} C_DIS
LIN {X -80.5911,Y -115.4583,Z 168,A -122.4783,B 9.9674,C 0.3422,E1 9.8834,E2 213.6785} C_DIS
LIN {X -77.0036,Y -117.8817,Z 168,A -120.7412,B 9.9673,C 0.3454,E1 9.8874,E2 211.9449} C_DIS
LIN {X -73.6332,Y -120.0152,Z 168,A -119.0683,B 9.9673,C 0.3467,E1 9.8914,E2 210.2657} C_DIS
LIN {X -69.9198,Y -122.216,Z 168,A -117.2958,B 9.9671,C 0.3487,E1 9.8957,E2 208.4912} C_DIS
LIN {X -66.1405,Y -124.3019,Z 168,A -115.6369,B 9.967,C 0.3531,E1 9.8997,E2 206.8453} C_DIS
LIN {X -62.8162,Y -126.0135,Z 168,A -114.0152,B 9.967,C 0.3528,E1 9.9038,E2 205.2105} C_DIS
LIN {X -59.1658,Y -127.7668,Z 168,A -112.5058,B 9.9668,C 0.3576,E1 9.9076,E2 203.7192} C_DIS
LIN {X -55.9614,Y -129.2024,Z 168,A -110.9193,B 9.9669,C 0.3557,E1 9.9117,E2 202.1119} C_DIS
LIN {X -51.7854,Y -130.9348,Z 168,A -109.1559,B 9.9668,C 0.3592,E1 9.9162,E2 200.3586} C_DIS
LIN {X -48.5577,Y -132.1659,Z 168,A -107.718,B 9.9668,C 0.3598,E1 9.92,E2 198.9162} C_DIS
LIN {X -44.5186,Y -133.5779,Z 168,A -106.0189,B 9.9667,C 0.3621,E1 9.9245,E2 197.2224} C_DIS
LIN {X -40.8183,Y -134.7554,Z 168,A -104.4084,B 9.9667,C 0.3627,E1 9.9288,E2 195.6076} C_DIS
LIN {X -37.5126,Y -135.7128,Z 168,A -102.941,B 9.9667,C 0.3621,E1 9.9327,E2 194.1312} C_DIS
LIN {X -33.6879,Y -136.7137,Z 168,A -101.2288,B 9.9667,C 0.3608,E1 9.9374,E2 192.405} C_DIS
LIN {X -30.3189,Y -137.4997,Z 168,A -100.0639,B 9.9665,C 0.3669,E1 9.9405,E2 191.2718} C_DIS
LIN {X -27.4563,Y -138.0998,Z 168,A -98.7914,B 9.9665,C 0.3656,E1 9.944,E2 189.9881} C_DIS
LIN {X -23.5393,Y -138.8203,Z 168,A -97.1542,B 9.9665,C 0.3659,E1 9.9485,E2 188.3483} C_DIS
LIN {X -20.6579,Y -139.2797,Z 168,A -95.9574,B 9.9665,C 0.3661,E1 9.9518,E2 187.1499} C_DIS
LIN {X -17.2232,Y -139.7452,Z 168,A -94.4386,B 9.9666,C 0.364,E1 9.9561,E2 185.6163} C_DIS
LIN {X -12.6105,Y -140.2377,Z 168,A -92.5256,B 9.9666,C 0.3637,E1 9.9614,E2 183.6992} C_DIS
LIN {X -8.0983,Y -140.5696,Z 168,A -90.689,B 9.9666,C 0.3639,E1 9.9665,E2 181.8625} C_DIS
LIN {X -3.3426,Y -140.7631,Z 168,A -88.9158,B 9.9665,C 0.3676,E1 9.9714,E2 180.11} C_DIS
LIN {X 0.5418,Y -140.8008,Z 168,A -87.304,B 9.9665,C 0.3667,E1 9.9759,E2 178.4933} C_DIS
LIN {X 0.5418,Y -140.8008,Z 168,A -87.304,B 9.9665,C 0.3667,E1 9.9759,E2 178.4933} C_DIS
Enddeposition()
LIN {X 0.956,Y -131.8451,Z 169,A -87.7498,B 9.9624,C 0.3209,E1 9.9698,E2 178.6752} C_DIS
Startdeposition()
$VEL.CP = VEL_PRINT
LIN {X -1.6121,Y -131.841,Z 169,A -89.1853,B 9.9622,C 0.3278,E1 9.9657,E2 180.15} C_DIS
LIN {X -4.823,Y -131.7617,Z 169,A -90.5732,B 9.9622,C 0.3276,E1 9.9618,E2 181.5375} C_DIS
LIN {X -8.0902,Y -131.6011,Z 169,A -91.9774,B 9.9622,C 0.3272,E1 9.9579,E2 182.9402} C_DIS
LIN {X -11.3135,Y -131.3634,Z 169,A -93.372,B 9.9622,C 0.3269,E1 9.954,E2 184.3341} C_DIS
LIN {X -14.5298,Y -131.0471,Z 169,A -94.7786,B 9.9622,C 0.3267,E1 9.9501,E2 185.7415} C_DIS
LIN {X -17.7463,Y -130.6511,Z 169,A -96.1851,B 9.9622,C 0.3263,E1 9.9462,E2 187.1484} C_DIS
LIN {X -20.8297,Y -130.1953,Z 169,A -97.5753,B 9.9622,C 0.3266,E1 9.9423,E2 188.5434} C_DIS
LIN {X -24.096,Y -129.6305,Z 169,A -99.0073,B 9.9622,C 0.3259,E1 9.9384,E2 189.9748} C_DIS
LIN {X -27.2666,Y -129.0003,Z 169,A -100.4256,B 9.9622,C 0.3255,E1 9.9345,E2 191.3951} C_DIS
LIN {X -30.4581,Y -128.2838,Z 169,A -101.8397,B 9.9623,C 0.3246,E1 9.9307,E2 192.8086} C_DIS
LIN {X -33.6047,Y -127.4954,Z 169,A -103.2486,B 9.9623,C 0.3237,E1 9.9269,E2 194.2177} C_DIS
LIN {X -36.645,Y -126.6551,Z 169,A -104.6364,B 9.9623,C 0.3231,E1 9.9231,E2 195.6078} C_DIS
LIN {X -39.7663,Y -125.7099,Z 169,A -106.0524,B 9.9623,C 0.322,E1 9.9193,E2 197.0239} C_DIS
LIN {X -42.8575,Y -124.6898,Z 169,A -107.4652,B 9.9624,C 0.3209,E1 9.9156,E2 198.4367} C_DIS
LIN {X -45.8988,Y -123.6027,Z 169,A -108.8654,B 9.9624,C 0.3196,E1 9.9119,E2 199.8366} C_DIS
LIN {X -48.9616,Y -122.4217,Z 169,A -110.2955,B 9.9625,C 0.3183,E1 9.9082,E2 201.2673} C_DIS
LIN {X -51.951,Y -121.1834,Z 169,A -111.7193,B 9.9625,C 0.3172,E1 9.9045,E2 202.6933} C_DIS
LIN {X -55.0252,Y -119.8186,Z 169,A -113.1808,B 9.9626,C 0.3156,E1 9.9008,E2 204.1548} C_DIS
LIN {X -57.8935,Y -118.4598,Z 169,A -114.568,B 9.9626,C 0.3142,E1 9.8973,E2 205.5429} C_DIS
LIN {X -60.7473,Y -117.0226,Z 169,A -115.9042,B 9.9627,C 0.3115,E1 9.894,E2 206.8729} C_DIS
LIN {X -62.8988,Y -115.8814,Z 169,A -117.1752,B 9.9627,C 0.3142,E1 9.8908,E2 208.1694} C_DIS
LIN {X -66.3609,Y -113.9344,Z 169,A -118.7857,B 9.9627,C 0.3097,E1 9.887,E2 209.7659} C_DIS
LIN {X -69.5866,Y -111.9929,Z 169,A -120.5524,B 9.9627,C 0.3099,E1 9.8827,E2 211.5481} C_DIS
LIN {X -73.2375,Y -109.6401,Z 169,A -122.3314,B 9.9629,C 0.305,E1 9.8786,E2 213.3138} C_DIS
LIN {X -75.9334,Y -107.7906,Z 169,A -123.7159,B 9.963,C 0.3021,E1 9.8754,E2 214.6938} C_DIS
LIN {X -78.5486,Y -105.9003,Z 169,A -125.1713,B 9.963,C 0.3008,E1 9.8721,E2 216.1552} C_DIS
LIN {X -81.1168,Y -103.9467,Z 169,A -126.6001,B 9.9631,C 0.2989,E1 9.869,E2 217.5869} C_DIS
LIN {X -84.258,Y -101.4166,Z 169,A -128.5218,B 9.9631,C 0.299,E1 9.8648,E2 219.5284} C_DIS
LIN {X -87.6676,Y -98.4847,Z 169,A -130.4234,B 9.9632,C 0.2944,E1 9.8608,E2 221.4231} C_DIS
LIN {X -90.9049,Y -95.5042,Z 169,A -132.4165,B 9.9633,C 0.2923,E1 9.8567,E2 223.4253} C_DIS
LIN {X -93.8187,Y -92.6439,Z 169,A -134.2206,B 9.9633,C 0.2893,E1 9.8531,E2 225.2323} C_DIS
LIN {X -97.133,Y -89.162,Z 169,A -136.1741,B 9.9636,C 0.2825,E1 9.8494,E2 227.1689} C_DIS
LIN {X -99.3174,Y -86.7222,Z 169,A -137.7597,B 9.9636,C 0.2825,E1 9.8465,E2 228.7732} C_DIS
LIN {X -102.0817,Y -83.4507,Z 169,A -139.434,B 9.9638,C 0.2751,E1 9.8435,E2 230.4244} C_DIS
LIN {X -104.4345,Y -80.4876,Z 169,A -141.3149,B 9.9638,C 0.2757,E1 9.8402,E2 232.3327} C_DIS
LIN {X -106.3946,Y -77.8776,Z 169,A -142.6644,B 9.9638,C 0.2712,E1 9.838,E2 233.6733} C_DIS
LIN {X -108.697,Y -74.6301,Z 169,A -144.3473,B 9.964,C 0.2663,E1 9.8353,E2 235.3496} C_DIS
LIN {X -110.5141,Y -71.912,Z 169,A -145.7644,B 9.9641,C 0.2629,E1 9.8331,E2 236.7656} C_DIS
LIN {X -112.229,Y -69.2057,Z 169,A -147.1832,B 9.9641,C 0.26,E1 9.831,E2 238.1867} C_DIS
LIN {X -113.9174,Y -66.3902,Z 169,A -148.6319,B 9.9643,C 0.2569,E1 9.829,E2 239.6372} C_DIS
LIN {X -115.5184,Y -63.5635,Z 169,A -149.9422,B 9.9644,C 0.2516,E1 9.8272,E2 240.9345} C_DIS
LIN {X -117.0189,Y -60.7544,Z 169,A -151.4726,B 9.9644,C 0.2507,E1 9.8252,E2 242.4814} C_DIS
LIN {X -118.4705,Y -57.8719,Z 169,A -152.8919,B 9.9645,C 0.2474,E1 9.8234,E2 243.9018} C_DIS
LIN {X -119.8514,Y -54.9544,Z 169,A -154.3119,B 9.9645,C 0.244,E1 9.8217,E2 245.3229} C_DIS
LIN {X -121.1676,Y -51.9877,Z 169,A -155.7411,B 9.9647,C 0.2406,E1 9.8201,E2 246.7533} C_DIS
LIN {X -122.3328,Y -49.182,Z 169,A -157.1095,B 9.9647,C 0.238,E1 9.8187,E2 248.1264} C_DIS
LIN {X -123.5745,Y -45.9739,Z 169,A -158.5994,B 9.9648,C 0.2339,E1 9.8172,E2 249.6146} C_DIS
LIN {X -124.6776,Y -42.8927,Z 169,A -160.0363,B 9.9649,C 0.2302,E1 9.8159,E2 251.0522} C_DIS
LIN {X -125.6924,Y -39.821,Z 169,A -161.3912,B 9.965,C 0.2255,E1 9.8147,E2 252.3999} C_DIS
LIN {X -126.6332,Y -36.72,Z 169,A -162.8845,B 9.965,C 0.2231,E1 9.8135,E2 253.9022} C_DIS
LIN {X -127.5015,Y -33.5819,Z 169,A -164.3188,B 9.9652,C 0.2195,E1 9.8125,E2 255.3376} C_DIS
LIN {X -128.2747,Y -30.4957,Z 169,A -165.7247,B 9.9652,C 0.216,E1 9.8115,E2 256.7451} C_DIS
LIN {X -128.9381,Y -27.5551,Z 169,A -167.0804,B 9.9652,C 0.2131,E1 9.8107,E2 258.1051} C_DIS
LIN {X -129.6192,Y -24.1552,Z 169,A -168.5782,B 9.9654,C 0.2086,E1 9.8099,E2 259.6005} C_DIS
LIN {X -130.1632,Y -21.03,Z 169,A -169.9742,B 9.9654,C 0.205,E1 9.8093,E2 260.9975} C_DIS
LIN {X -130.6413,Y -17.8211,Z 169,A -171.4425,B 9.9655,C 0.202,E1 9.8087,E2 262.4714} C_DIS
LIN {X -130.9595,Y -15.2965,Z 169,A -172.6822,B 9.9655,C 0.2011,E1 9.8083,E2 263.7257} C_DIS
LIN {X -131.3635,Y -11.3114,Z 169,A -174.3028,B 9.9657,C 0.194,E1 9.8079,E2 265.3306} C_DIS
LIN {X -131.5852,Y -8.3479,Z 169,A -175.6673,B 9.9657,C 0.1915,E1 9.8076,E2 266.7025} C_DIS
LIN {X -131.7604,Y -4.8569,Z 169,A -177.3063,B 9.9657,C 0.1891,E1 9.8074,E2 268.3541} C_DIS
LIN {X -131.8522,Y -0.2351,Z 169,A -179.2756,B 9.9659,C 0.1826,E1 9.8074,E2 270.3169} C_DIS
LIN {X -131.8106,Y 3.2331,Z 169,A 179.2661,B 9.9659,C 0.1774,E1 9.8074,E2 271.768} C_DIS
LIN {X -131.691,Y 6.4648,Z 169,A 177.8372,B 9.9661,C 0.1737,E1 9.8076,E2 273.1982} C_DIS
LIN {X -131.4928,Y 9.6925,Z 169,A 176.4182,B 9.9661,C 0.1698,E1 9.8079,E2 274.6174} C_DIS
LIN {X -131.2196,Y 12.8752,Z 169,A 175.0071,B 9.9661,C 0.1662,E1 9.8082,E2 276.0298} C_DIS
LIN {X -130.8545,Y 16.1769,Z 169,A 173.5523,B 9.9662,C 0.1622,E1 9.8087,E2 277.4845} C_DIS
LIN {X -130.4257,Y 19.3355,Z 169,A 172.1345,B 9.9662,C 0.1587,E1 9.8093,E2 278.9047} C_DIS
LIN {X -129.9077,Y 22.5543,Z 169,A 170.701,B 9.9664,C 0.1549,E1 9.8099,E2 280.3388} C_DIS
LIN {X -129.3752,Y 25.4316,Z 169,A 169.3387,B 9.9664,C 0.1528,E1 9.8106,E2 281.7102} C_DIS
LIN {X -128.7462,Y 28.4437,Z 169,A 167.9351,B 9.9664,C 0.1501,E1 9.8115,E2 283.1203} C_DIS
LIN {X -127.8982,Y 32.0381,Z 169,A 166.4151,B 9.9665,C 0.1441,E1 9.8125,E2 284.6286} C_DIS
LIN {X -127.0859,Y 35.122,Z 169,A 164.9952,B 9.9665,C 0.1408,E1 9.8135,E2 286.051} C_DIS
LIN {X -126.2093,Y 38.1525,Z 169,A 163.5934,B 9.9666,C 0.1374,E1 9.8146,E2 287.4549} C_DIS
LIN {X -125.2091,Y 41.3157,Z 169,A 162.1568,B 9.9666,C 0.1333,E1 9.8158,E2 288.8895} C_DIS
LIN {X -124.1582,Y 44.374,Z 169,A 160.7324,B 9.9667,C 0.1297,E1 9.8172,E2 290.3145} C_DIS
LIN {X -123.0187,Y 47.4415,Z 169,A 159.4681,B 9.9667,C 0.1231,E1 9.8184,E2 291.559} C_DIS
LIN {X -121.6838,Y 50.7663,Z 169,A 157.6188,B 9.9667,C 0.1239,E1 9.8204,E2 293.4407} C_DIS
LIN {X -119.8703,Y 54.9134,Z 169,A 155.7203,B 9.9669,C 0.1175,E1 9.8225,E2 295.3291} C_DIS
LIN {X -118.4885,Y 57.8353,Z 169,A 154.2979,B 9.9669,C 0.114,E1 9.8242,E2 296.752} C_DIS
LIN {X -117.0357,Y 60.7224,Z 169,A 152.93,B 9.9669,C 0.1097,E1 9.8259,E2 298.1143} C_DIS
LIN {X -115.5109,Y 63.5769,Z 169,A 151.4471,B 9.9669,C 0.1074,E1 9.8279,E2 299.6045} C_DIS
LIN {X -113.9221,Y 66.3821,Z 169,A 150.0174,B 9.967,C 0.1043,E1 9.8299,E2 301.0361} C_DIS
LIN {X -112.2461,Y 69.1778,Z 169,A 148.5834,B 9.967,C 0.1011,E1 9.832,E2 302.4706} C_DIS
LIN {X -110.5216,Y 71.9004,Z 169,A 147.1749,B 9.967,C 0.0977,E1 9.8341,E2 303.8786} C_DIS
LIN {X -108.7542,Y 74.5467,Z 169,A 145.7611,B 9.9671,C 0.0949,E1 9.8363,E2 305.2945} C_DIS
Enddeposition()
END
